// TwinCAT 3 PLC project PShEll_UniversalBlocks
// Title: PShEll Universal Blocks
// Company: Precision Systems Engineering
// Author: Control Systems Design Department
// ProjectVersion: 1.0.1.1
// Description: PSE Shell - Automation Software Development Kit
// ProgramVersion: 3.1.4023.0
// libraries:
//   CmpBitmapPool, * (System)
//   JS_MC_REF, * (Jenny Science AG)
//   Recipe Management, * (System)
//   Tc2_EtherCAT, * (Beckhoff Automation GmbH)
//   Tc2_IoFunctions, * (Beckhoff Automation GmbH)
//   Tc2_MC2, * (Beckhoff Automation GmbH)
//   Tc2_Standard, * (Beckhoff Automation GmbH)
//   Tc2_SUPS, * (Beckhoff Automation GmbH)
//   Tc2_System, * (Beckhoff Automation GmbH)
//   Tc2_SystemCX, * (Beckhoff Automation GmbH)
//   Tc2_TcpIp, * (Beckhoff Automation GmbH)
//   Tc2_Utilities, * (Beckhoff Automation GmbH)
//   Tc3_EventLogger, * (Beckhoff Automation GmbH)
//   Tc3_McCollisionAvoidance, * (Beckhoff Automation GmbH)
//   Tc3_McCompensations, * (Beckhoff Automation GmbH)
//   Tc3_McCoordinatedMotion, * (Beckhoff Automation GmbH)
//   Tc3_Module, * (Beckhoff Automation GmbH)
//   Tc3_XTS_Utility, * (Beckhoff Automation GmbH)
//   VisuDialogs, * (System)
//   VisuUserMgmt, * (System)
//   Tc2_Math,3.3.1.0,Beckhoff Automation GmbH
//   VisuSymbols,3.5.10.0,System
// project tree:
//   DUTs/Libs/Alarms/AlarmControler/ E_AlarmControlerState.TcDUT
//   DUTs/Libs/Alarms/VisuEvents/ E_EventType.TcDUT, ST_BaseEvent.TcDUT, ST_Event.TcDUT
//   DUTs/Libs/Axis/Universal Axis/ E_AxisJogDirection.TcDUT, E_AxisState.TcDUT, E_AxisStateInit.TcDUT, E_AxisStatePlcOpen.TcDUT
//   DUTs/Libs/Communication/TcpIp/ E_TcpIpDeviceState.TcDUT, E_TcpIpDeviceStateRecive.TcDUT, E_TcpIpDeviceStateSend.TcDUT, E_TcpIpServerStateRunning.TcDUT, ST_TcpBufferData.TcDUT
//   DUTs/Libs/Cylinder/Universal Cylinder/ E_CylinderError.TcDUT, E_CylinderState.TcDUT, E_CylinderStateGo.TcDUT
//   DUTs/Libs/Digital Devices/Digital Input/ E_DigitalInputExState.TcDUT
//   DUTs/Libs/Digital Devices/Lamp Indicator/ E_LampState.TcDUT
//   DUTs/Libs/Fixtures/UniversalFixture/ E_UniversalFixtureConnectionType.TcDUT, E_UniversalFixtureSampleResult.TcDUT, E_UniversalFixtureState.TcDUT, E_UniversalFixtureStateAbort.TcDUT, E_UniversalFixtureStateInit.TcDUT, E_UniversalFixtureStateMeasure.TcDUT, E_UniversalFixtureStateReset.TcDUT
//   DUTs/Libs/Platform/Common/ ST_UniversalPlatform.TcDUT
//   DUTs/Libs/Platform/Universal Machine/ E_MachineCtrlState.TcDUT
//   DUTs/Libs/Platform/Universal Safety/ E_SafetyCtrlState.TcDUT
//   DUTs/Libs/Platform/Universal Visu/ E_VisuCtrlAlarmControlState.TcDUT, E_VisuCtrlAxisImgType.TcDUT, E_VisuCtrlAxisJogMode.TcDUT, E_VisuCtrlCylinderImgType.TcDUT, E_VisuCtrlNavBarState.TcDUT, E_VisuCtrlPageState.TcDUT, E_VisuCtrlRecipeParameterType.TcDUT, E_VisuCtrlRecipesManagerState.TcDUT, E_VisuCtrlRobotImgType.TcDUT, E_VisuCtrlSingleAxisState.TcDUT, E_VisuCtrlSingleCylinderState.TcDUT, E_VisuCtrlSingleRobotState.TcDUT, E_VisuCtrUniversalMachineState.TcDUT, ST_VisuCtrlAxisFrame.TcDUT, ST_VisuCtrlCylinderFrame.TcDUT, ST_VisuCtrlFixtureFrame.TcDUT, ST_VisuCtrlInputFrame.TcDUT, ST_VisuCtrlOutputFrame.TcDUT, ST_VisuCtrlRecipeParameter.TcDUT, ST_VisuCtrlRecipesManager.TcDUT, ST_VisuCtrlRobotFrame.TcDUT, ST_VisuCtrlUnitFrame.TcDUT
//   DUTs/Libs/Robots/Mitsubishi/CR800/EtherCAT Registers/ ST_CR800EthercatData.TcDUT
//   DUTs/Libs/Robots/Mitsubishi/CR800/ E_CR800Error.TcDUT, ST_CR800UserDefinedArea.TcDUT
//   DUTs/Libs/Robots/Mitsubishi/CR800/StateMachine/ E_CR800State.TcDUT, E_CR800StateAborting.TcDUT, E_CR800StateCommandExchange.TcDUT, E_CR800StateCyclePausing.TcDUT, E_CR800StateCycleStopping.TcDUT, E_CR800StateDoingRequest.TcDUT, E_CR800StateHoming.TcDUT, E_CR800StateInitializing.TcDUT, E_CR800StateSendPosition.TcDUT
//   DUTs/Libs/Robots/Mitsubishi/ E_RobotActions.TcDUT, E_RobotSystemActions.TcDUT
//   DUTs/Libs/Utilities/CSV Data Exchanger/ E_CSVDataExchangerCountColumnsState.TcDUT, E_CSVDataExchangerInitState.TcDUT, E_CSVDataExchangerInsertIntoTableState.TcDUT, E_CSVDataExchangerSelectAllState.TcDUT, E_CSVDataExchangerSelectRowState.TcDUT, E_CSVDataExchangerSetNewPathState.TcDUT, E_CSVDataExchangerState.TcDUT, ST_CSV_Record.TcDUT
//   DUTs/Libs/Utilities/File Logger/ E_FileLoggerAddLogsState.TcDUT, E_FileLoggerInitState.TcDUT, E_FileLoggerSetNewPathState.TcDUT, E_FileLoggerState.TcDUT
//   DUTs/Libs/Utilities/Recipe Manager/ E_RecipesManagerReturns.TcDUT, E_RecipesManagerState.TcDUT, E_RecipesManagerStateBackup.TcDUT, E_RecipesManagerStateCreateRemove.TcDUT, E_RecipesManagerStateInit.TcDUT, E_RecipesManagerStateReload.TcDUT
//   DUTs/Libs/Utilities/TXT Data Exchanger/ E_TXTDataExchangerAddLogsState.TcDUT, E_TXTDataExchangerInitState.TcDUT, E_TXTDataExchangerSearchForFileState.TcDUT, E_TXTDataExchangerSetNewPathState.TcDUT, E_TXTDataExchangerState.TcDUT
//   DUTs/Libs/Vision/Cognex/ E_CognexCameraGetConnectionStatus.TcDUT, E_CognexCameraGetExprStatus.TcDUT, E_CognexCameraGetFileListStatus.TcDUT, E_CognexCameraGetFileStatus.TcDUT, E_CognexCameraGetJobStatus.TcDUT, E_CognexCameraGetOnlineStatus.TcDUT, E_CognexCameraGetPositionState.TcDUT, E_CognexCameraGetPositionStatus.TcDUT, E_CognexCameraGetValueEasyBuilderStatus.TcDUT, E_CognexCameraGetValueSpreadsheetStatus.TcDUT, E_CognexCameraGetValuesState.TcDUT, E_CognexCameraGetValuesStatus.TcDUT, E_CognexCameraGetValueStatus.TcDUT, E_CognexCameraImageTriggerStatus.TcDUT, E_CognexCameraInitState.TcDUT, E_CognexCameraLoadFileStatus.TcDUT, E_CognexCameraMethodState.TcDUT, E_CognexCameraPutLiveStatus.TcDUT, E_CognexCameraPutPortnumStatus.TcDUT, E_CognexCameraPutTimeoutStatus.TcDUT, E_CognexCameraPutUpdateStatus.TcDUT, E_CognexCameraPutWatchStatus.TcDUT, E_CognexCameraResetSystemStatus.TcDUT, E_CognexCameraSetJobStatus.TcDUT, E_CognexCameraSetOnlineStatus.TcDUT, E_CognexCameraState.TcDUT, E_CognexCameraStoreFileStatus.TcDUT
//   DUTs/Machine/Machine Control/ E_MachineCtrlStateInit.TcDUT, E_MachineCtrlStateUninitialized.TcDUT
//   DUTs/Machine/Shell API/ ST_Shell.TcDUT, ST_ShellFlags.TcDUT, ST_ShellPlatform.TcDUT, ST_ShellRecipeData.TcDUT
//   DUTs/Platform/Universal Visu/ ST_VisuCtrlRobotFrame.TcDUT (not stored)
//   / GlobalTextList.TcGTLO, Test.TcTTO, Visualization Manager.TcVMO (not stored), VISU_TASK.TcTTO
//   GVLs/ GVL.TcGVL
//   POUs/Libs/0_Checks/Checks/ CheckBounds.TcPOU, CheckDivDInt.TcPOU, CheckDivLInt.TcPOU, CheckDivLReal.TcPOU, CheckDivReal.TcPOU, CheckPointer.TcPOU, CheckRangeSigned.TcPOU, CheckRangeUnsigned.TcPOU, P_Checks.TcPOU
//   POUs/Libs/0_Checks/ GVL_Checks.TcGVL
//   POUs/Libs/Alarms/AlarmControler/ FB_AlarmControler.TcPOU, I_AlarmControler.TcIO
//   POUs/Libs/Alarms/VisuEvents/ FB_VisuEventsHandling.TcPOU, LDT_TO_STRING.TcPOU
//   POUs/Libs/Axis/ FB_AxisServo.TcPOU, FB_UniversalAxis.TcPOU, I_UniversalAxis.TcIO
//   POUs/Libs/Communication/TcpIp/ FUN_StringToTcpBufferData.TcPOU, FUN_TcpBufferDataToString.TcPOU
//   POUs/Libs/Communication/TcpIp/Tcp Buffer/ FB_TcpBuffer.TcPOU
//   POUs/Libs/Communication/TcpIp/Tcp Client/ FB_TcpClient.TcPOU
//   POUs/Libs/Communication/TcpIp/Tcp Device/ FB_TcpDevice.TcPOU, I_TcpDevice.TcIO
//   POUs/Libs/Communication/TcpIp/Tcp Server/ FB_TcpServer.TcPOU
//   POUs/Libs/Cylinder/Double Coil Cylinder/ FB_DoubleCoilCylinder.TcPOU, FB_DoubleCoilCylinder2.TcPOU
//   POUs/Libs/Cylinder/Single Coil Cylinder/ FB_SingleCoilCylinder.TcPOU, FB_SingleCoilCylinder2.TcPOU
//   POUs/Libs/Cylinder/Universal Cylinder/ FB_UniversalCylinder.TcPOU, I_UniversalCylinder.TcIO
//   POUs/Libs/Digital Devices/Digital Device/ FB_DigitalDevice.TcPOU, I_DigitalDevice.TcIO
//   POUs/Libs/Digital Devices/Digital Input/ FB_DigitalInput.TcPOU, FB_DigitalInputExt.TcPOU, I_DigitalInput.TcIO
//   POUs/Libs/Digital Devices/Digital Output/ FB_DigitalOutput.TcPOU, I_DigitalOutput.TcIO
//   POUs/Libs/Digital Devices/Lamp Indicator/ FB_Lamp.TcPOU, I_Lamp.TcIO
//   POUs/Libs/Fixtures/ FB_UniversalFixture.TcPOU, I_UniversalFixture.TcIO
//   POUs/Libs/Platform/Universal Machine/ FB_UniversalMachine.TcPOU, I_UniversalMachine.TcIO
//   POUs/Libs/Platform/Universal Safety/ FB_UniversalSafety.TcPOU, I_UniversalSafety.TcIO
//   POUs/Libs/Platform/Universal Visu/ FB_UniversalVisu.TcPOU, F_CloseDialog.TcPOU, F_OpenDialog.TcPOU
//   POUs/Libs/Robots/Mitsubishi/ FB_CR800EtherCAT.TcPOU, I_CR800EtherCAT.TcIO
//   POUs/Libs/Utilities/Beckhoff UPS/CX2xxx/ FB_UpsCx2xxx.TcPOU
//   POUs/Libs/Utilities/Beckhoff UPS/CX5xxx/ FB_UpsCx50xx.TcPOU, FB_UpsCx51xx.TcPOU, FB_UpsCx5xxx.TcPOU, I_BeckhoffUpsCX5xxx.TcIO
//   POUs/Libs/Utilities/Beckhoff UPS/Universal CX/ FB_UniversalCxUps.TcPOU, I_UniversalCxUps.TcIO
//   POUs/Libs/Utilities/CSV Data Exchanger/ FB_CSVDataExchanger.TcPOU, I_CSVDataExchanger.TcIO
//   POUs/Libs/Utilities/File Logger/ FB_FileLogger.TcPOU, I_FileLogger.TcIO
//   POUs/Libs/Utilities/Math/ FUN_Ceil.TcPOU
//   POUs/Libs/Utilities/Recipes Manager/ FB_RecipeParameter.TcPOU, FB_RecipesControler.TcPOU, I_RecipeParameter.TcIO, I_RecipesManager.TcIO
//   POUs/Libs/Utilities/StringMerge/ FUN_MergeLongStrings10.TcPOU, FUN_MergeStrings10.TcPOU, FUN_MergeStrings3.TcPOU, FUN_MergeStrings4.TcPOU, FUN_MergeStrings5.TcPOU, FUN_MergeStrings6.TcPOU
//   POUs/Libs/Utilities/Systemtime to String/ FUN_TimestructToDate.TcPOU, FUN_TimestructToTime.TcPOU
//   POUs/Libs/Utilities/TXT Data Exchanger/ FB_TXTDataExchanger.TcPOU, I_TXTDataExchanger.TcIO
//   POUs/Libs/Vision/Cognex/ FB_CognexCamera.TcPOU, I_CognexCamera.TcIO
//   POUs/Machine/Alarm Control/ PRG_AlarmControl.TcPOU
//   POUs/Machine/Machine Control/ FB_MachineControl.TcPOU, I_MachineControl.TcIO, PRG_MachineControl.TcPOU
//   POUs/Machine/Recipes Manager/ PRG_RecipesManager.TcPOU
//   POUs/Machine/Visu Control/ FB_VisuControl.TcPOU, F_CloseDialog_1.TcPOU, F_OpenDialog_1.TcPOU, PRG_VisuControl.TcPOU
//   VISUs/Alarms/ EventTable.TcVIS, EventTableNew.TcVIS (not stored), SingleEvent.TcVIS (not stored)
//   VISUs/Alarms/Image Pools/ IP_EventSeverity.TcIPO (not stored), IP_EventType.TcIPO (not stored)
//   VISUs/Alarms/Text Lists/ TL_EventServerity.TcTLO (not stored), TL_EventType.TcTLO (not stored)
//   VISUs/Headers/ Header.TcVIS, HeaderWinCE.TcVIS
//   VISUs/Headers/Image Pools/ IPHeader.TcIPO (not stored)
//   VISUs/Headers/Text Lists/ TL_HeaderMachineState.TcTLO
//   VISUs/ Main.TcVIS
//   VISUs/Manual/Image Pools/ IPAxis.TcIPO (not stored), IPCylinder.TcIPO (not stored), IPRobots.TcIPO (not stored)
//   VISUs/Manual/ SingleAxis.TcVIS, SingleFixture.TcVIS, SingleAxisJogInching.TcVIS, SingleAxisJogContinous.TcVIS, SingleAxisJogInchingModulo.TcVIS, SingleAxisJogStandardSlow.TcVIS, SingleAxisJogStandardFlast.TcVIS, SingleCylinder.TcVIS, SingleDigitalInput.TcVIS, SingleRobot.TcVIS, SingleSafeOutput.TcVIS (excluded from build), SingleSafeInput.TcVIS (excluded from build), SingleDigitalOutput.TcVIS
//   VISUs/Manual/Text Lists/ TL_ModeSwitchState.TcTLO, TL_SingleAxisJogMode.TcTLO, TL_SingleCylinderState.TcTLO, TL_SingleAxisState.TcTLO, TL_SingleRobotState.TcTLO
//   VISUs/Navigation/ NavBarAuto.TcVIS, NavBarAuxilary.TcVIS, NavBarEmpty.TcVIS, NavBarInitializing.TcVIS, NavBarManual.TcVIS, NavBarUninitialized.TcVIS, NavBarUtilities.TcVIS
//   VISUs/Pages/ PageInitializing.TcVIS, PageXtsEnviroment.TcVIS (excluded from build), PageAborting.TcVIS, PageAlarms.TcVIS, PageManualCylinders.TcVIS, PageManualRobots.TcVIS, PageManualInputs.TcVIS, PageManualAxis.TcVIS, PageManualOutputs.TcVIS, PageManualSafety.TcVIS (excluded from build), PageReadyInitialized.TcVIS, PageRecipesManager.TcVIS, PageReset.TcVIS, PageSwitchMode.TcVIS, PageXtsDiagnostic.TcVIS (excluded from build)
//   VISUs/Recipes/ SingleRecipesParameterTypeBool.TcVIS, SingleRecipesParameterTypeInteger.TcVIS, SingleRecipesParameterTypeReal.TcVIS, SingleRecipesParameterTypeString.TcVIS
//   VISUs/Recipes/Text Lists/ TL_RecipesManagerReturns.TcTLO, TL_RecipesManagerStatus.TcTLO
// real-time tasks:
//   TASK SampleTests Task: cycle T#10ms, priority 20, ADS port 350
//   TASK UniversalBlocks Task: cycle T#10ms, priority 22, ADS port 351
//   TASK Job Task: cycle default, priority 32
//   TASK VISU_TASK: cycle T#200000us, priority 30, ADS port 352
//   TASK XTS Task 1: cycle T#250us, priority 1, ADS port 353
//   TASK TestAlarms: cycle T#2ms, priority 21, ADS port 354
//   TASK Test: cycle T#10ms, priority 23, ADS port 355
// motion (NC):
//   TASK NC-Task 1 SAF: cycle T#2ms, priority 4, ADS port 501
//   TASK NC-Task 1 SVB: cycle T#10ms, priority 8, ADS port 511
//   AXIS Faulhaber_LM1247_PNP2_1 (id 11)
//     Dynamic: AccelerationMaximum=1000000, DecelerationMaximum=1000000, Acceleration=5000, Deceleration=5000, Jerk=10000
//     Velo: RefSearch=25, RefSync=15, SlowManual=10, FastManual=25
//     PositionAreaControl: Enable=false
//     TargetPosControl: Range=0.1, Time=0.01
//     OtherSettings: AllowMotionCmdToSlave=true, PulseDistancePos=10, PulseDistanceNeg=10
//     encoder EncType=19
//       EncPara: ScaleFactorNumerator=0.001, MaxCount=#xffffffff
//         SoftEndMinControl: Enable=true, Range=-80
//         SoftEndMaxControl: Enable=true, Range=80
//     drive DrvType=16
//       DrvPara: MaxCount=#xffffffff
//         Analog: VeloReferenz=2000, TorqueSetpointScale=10, ScaleFactorActTorque=0.1
//         TimeComp: TaskDelayCycles=1
//     controller CtrType=3
//       CtrPara: PriorControlFactor=1
//         PosDiffControl: Enable=false
//         PID: PosTn=0.1
//         Observer: BandWidth=20
//   AXIS Faulhaber_LM1247_PNP2_2 (id 7)
//     Dynamic: AccelerationMaximum=1000000, DecelerationMaximum=1000000, Acceleration=5000, Deceleration=5000, Jerk=10000
//     Velo: RefSearch=25, RefSync=15, SlowManual=10, FastManual=25
//     PositionAreaControl: Enable=false
//     TargetPosControl: Range=0.1, Time=0.01
//     OtherSettings: AllowMotionCmdToSlave=true, PulseDistancePos=10, PulseDistanceNeg=10
//     encoder EncType=19
//       EncPara: ScaleFactorNumerator=0.001, MaxCount=#xffffffff
//         SoftEndMinControl: Enable=true, Range=-80
//         SoftEndMaxControl: Enable=true, Range=80
//     drive DrvType=16
//       DrvPara: MaxCount=#xffffffff
//         Analog: VeloReferenz=2000, TorqueSetpointScale=10, ScaleFactorActTorque=0.1
//         TimeComp: TaskDelayCycles=1
//     controller CtrType=3
//       CtrPara: PriorControlFactor=1
//         PosDiffControl: Enable=false
//         PID: PosTn=0.1
//         Observer: BandWidth=20
//   AXIS Faulhaber_LM1247_PNP2_3 (id 8)
//     Dynamic: AccelerationMaximum=1000000, DecelerationMaximum=1000000, Acceleration=5000, Deceleration=5000, Jerk=10000
//     Velo: RefSearch=25, RefSync=15, SlowManual=10, FastManual=25
//     PositionAreaControl: Enable=false
//     TargetPosControl: Range=0.1, Time=0.01
//     OtherSettings: AllowMotionCmdToSlave=true, PulseDistancePos=10, PulseDistanceNeg=10
//     encoder EncType=19
//       EncPara: ScaleFactorNumerator=0.001, MaxCount=#xffffffff
//         SoftEndMinControl: Enable=true, Range=-80
//         SoftEndMaxControl: Enable=true, Range=80
//     drive DrvType=16
//       DrvPara: MaxCount=#xffffffff
//         Analog: VeloReferenz=2000, TorqueSetpointScale=10, ScaleFactorActTorque=0.1
//         TimeComp: TaskDelayCycles=1
//     controller CtrType=3
//       CtrPara: PriorControlFactor=1
//         PosDiffControl: Enable=false
//         PID: PosTn=0.1
//         Observer: BandWidth=20
//   AXIS Faulhaber_LM1247_PNP2_4 (id 9)
//     Dynamic: AccelerationMaximum=1000000, DecelerationMaximum=1000000, Acceleration=5000, Deceleration=5000, Jerk=10000
//     Velo: RefSearch=25, RefSync=15, SlowManual=10, FastManual=25
//     PositionAreaControl: Enable=false
//     TargetPosControl: Range=0.1, Time=0.01
//     OtherSettings: AllowMotionCmdToSlave=true, PulseDistancePos=10, PulseDistanceNeg=10
//     encoder EncType=19
//       EncPara: ScaleFactorNumerator=0.001, MaxCount=#xffffffff
//         SoftEndMinControl: Enable=true, Range=-80
//         SoftEndMaxControl: Enable=true, Range=80
//     drive DrvType=16
//       DrvPara: MaxCount=#xffffffff
//         Analog: VeloReferenz=2000, TorqueSetpointScale=10, ScaleFactorActTorque=0.1
//         TimeComp: TaskDelayCycles=1
//     controller CtrType=3
//       CtrPara: PriorControlFactor=1
//         PosDiffControl: Enable=false
//         PID: PosTn=0.1
//         Observer: BandWidth=20
//   AXIS Faulhaber_LM1247_PNP2_5 (id 10)
//     Dynamic: AccelerationMaximum=1000000, DecelerationMaximum=1000000, Acceleration=5000, Deceleration=5000, Jerk=10000
//     Velo: RefSearch=25, RefSync=15, SlowManual=10, FastManual=25
//     PositionAreaControl: Enable=false
//     TargetPosControl: Range=0.1, Time=0.01
//     OtherSettings: AllowMotionCmdToSlave=true, PulseDistancePos=10, PulseDistanceNeg=10
//     encoder EncType=19
//       EncPara: ScaleFactorNumerator=0.001, MaxCount=#xffffffff
//         SoftEndMinControl: Enable=true, Range=-80
//         SoftEndMaxControl: Enable=true, Range=80
//     drive DrvType=16
//       DrvPara: MaxCount=#xffffffff
//         Analog: VeloReferenz=2000, TorqueSetpointScale=10, ScaleFactorActTorque=0.1
//         TimeComp: TaskDelayCycles=1
//     controller CtrType=3
//       CtrPara: PriorControlFactor=1
//         PosDiffControl: Enable=false
//         PID: PosTn=0.1
//         Observer: BandWidth=20
//   AXIS Faulhaber_LM1247_PNP2_6 (id 12)
//     Dynamic: AccelerationMaximum=1000000, DecelerationMaximum=1000000, Acceleration=5000, Deceleration=5000, Jerk=10000
//     Velo: RefSearch=25, RefSync=15, SlowManual=10, FastManual=25
//     PositionAreaControl: Enable=false
//     TargetPosControl: Range=0.1, Time=0.01
//     OtherSettings: AllowMotionCmdToSlave=true, PulseDistancePos=10, PulseDistanceNeg=10
//     encoder EncType=19
//       EncPara: ScaleFactorNumerator=0.001, MaxCount=#xffffffff
//         SoftEndMinControl: Enable=true, Range=-80
//         SoftEndMaxControl: Enable=true, Range=80
//     drive DrvType=16
//       DrvPara: MaxCount=#xffffffff
//         Analog: VeloReferenz=2000, TorqueSetpointScale=10, ScaleFactorActTorque=0.1
//         TimeComp: TaskDelayCycles=1
//     controller CtrType=3
//       CtrPara: PriorControlFactor=1
//         PosDiffControl: Enable=false
//         PID: PosTn=0.1
//         Observer: BandWidth=20
//   AXIS Faulhaber_LM1247_PNP1_2 (id 14)
//     Dynamic: AccelerationMaximum=1000000, DecelerationMaximum=1000000, Acceleration=5000, Deceleration=5000, Jerk=10000
//     Velo: RefSearch=25, RefSync=25, SlowManual=10, FastManual=25
//     PositionAreaControl: Enable=false
//     TargetPosControl: Range=0.1, Time=0.01
//     OtherSettings: AllowMotionCmdToSlave=true, PulseDistancePos=10, PulseDistanceNeg=10
//     encoder EncType=19
//       EncPara: ScaleFactorNumerator=0.001, MaxCount=#xffffffff
//         SoftEndMinControl: Enable=true, Range=-80
//         SoftEndMaxControl: Enable=true, Range=80
//     drive DrvType=16
//       DrvPara: MaxCount=#xffffffff
//         Analog: VeloReferenz=2000, TorqueSetpointScale=10, ScaleFactorActTorque=0.1
//         TimeComp: TaskDelayCycles=1
//     controller CtrType=3
//       CtrPara: PriorControlFactor=1
//         PosDiffControl: Enable=false
//         PID: PosTn=0.1
//         Observer: BandWidth=20
//   AXIS Faulhaber_LM1247_PNP1_6 (id 13)
//     Dynamic: AccelerationMaximum=1000000, DecelerationMaximum=1000000, Acceleration=5000, Deceleration=5000, Jerk=10000
//     Velo: RefSearch=25, RefSync=25, SlowManual=10, FastManual=25
//     PositionAreaControl: Enable=false
//     TargetPosControl: Range=0.1, Time=0.01
//     OtherSettings: AllowMotionCmdToSlave=true, PulseDistancePos=10, PulseDistanceNeg=10
//     encoder EncType=1
//       EncPara: ScaleFactorNumerator=0.001
//         SoftEndMinControl: Enable=true, Range=-80
//         SoftEndMaxControl: Enable=true, Range=80
//     drive DrvType=5
//       Analog: VeloReferenz=10, TorqueSetpointScale=10, ScaleFactorActTorque=0.1
//       TimeComp: TaskDelayCycles=1
//     controller CtrType=3
//       CtrPara: PriorControlFactor=1
//         PosDiffControl: Enable=false
//         PID: PosTn=0.1
//         Observer: BandWidth=20
//   AXIS Mover Axis 1 (id 15)
//     General: UnitFlags=#x00000004
//     Dynamic: AccelerationMaximum=80000, DecelerationMaximum=80000, Acceleration=20000, Deceleration=20000, Jerk=200000
//     Velo: Maximum=4000
//     PositionAreaControl: Enable=false
//     TargetPosControl: Enable=false
//     OtherSettings: AllowMotionCmdToSlave=true, AllowMotionCmdToExtSetGenAxis=true
//     encoder EncType=28
//       EncPara: ModuloFactor=2500, ToleranceWndModuloStart=0.2, MaxCount=#xffffffff
//     drive DrvType=22
//       DrvPara: MaxCount=#xffffffff, DriveControlDWord=#x00000100
//         Analog: VeloReferenz=4200, TorqueSetpointScale=10
//         TimeComp: TaskDelayCycles=1
//     controller CtrType=1
//       CtrPara: PriorControlFactor=1
//         PosDiffControl: Range=10
//         Observer: BandWidth=20
//   AXIS Mover Axis 2 (id 16)
//     General: UnitFlags=#x00000004
//     Dynamic: AccelerationMaximum=80000, DecelerationMaximum=80000, Acceleration=20000, Deceleration=20000, Jerk=200000
//     Velo: Maximum=4000
//     PositionAreaControl: Enable=false
//     TargetPosControl: Enable=false
//     OtherSettings: AllowMotionCmdToSlave=true, AllowMotionCmdToExtSetGenAxis=true
//     encoder EncType=28
//       EncPara: ModuloFactor=2500, ToleranceWndModuloStart=0.2, MaxCount=#xffffffff
//     drive DrvType=22
//       DrvPara: MaxCount=#xffffffff, DriveControlDWord=#x00000100
//         Analog: VeloReferenz=4200, TorqueSetpointScale=10
//         TimeComp: TaskDelayCycles=1
//     controller CtrType=1
//       CtrPara: PriorControlFactor=1
//         PosDiffControl: Range=10
//         Observer: BandWidth=20
//   AXIS Mover Axis 3 (id 17)
//     General: UnitFlags=#x00000004
//     Dynamic: AccelerationMaximum=80000, DecelerationMaximum=80000, Acceleration=20000, Deceleration=20000, Jerk=200000
//     Velo: Maximum=4000
//     PositionAreaControl: Enable=false
//     TargetPosControl: Enable=false
//     OtherSettings: AllowMotionCmdToSlave=true, AllowMotionCmdToExtSetGenAxis=true
//     encoder EncType=28
//       EncPara: ModuloFactor=2500, ToleranceWndModuloStart=0.2, MaxCount=#xffffffff
//     drive DrvType=22
//       DrvPara: MaxCount=#xffffffff, DriveControlDWord=#x00000100
//         Analog: VeloReferenz=4200, TorqueSetpointScale=10
//         TimeComp: TaskDelayCycles=1
//     controller CtrType=1
//       CtrPara: PriorControlFactor=1
//         PosDiffControl: Range=10
//         Observer: BandWidth=20
//   AXIS Mover Axis 4 (id 18)
//     General: UnitFlags=#x00000004
//     Dynamic: AccelerationMaximum=80000, DecelerationMaximum=80000, Acceleration=20000, Deceleration=20000, Jerk=200000
//     Velo: Maximum=4000
//     PositionAreaControl: Enable=false
//     TargetPosControl: Enable=false
//     OtherSettings: AllowMotionCmdToSlave=true, AllowMotionCmdToExtSetGenAxis=true
//     encoder EncType=28
//       EncPara: ModuloFactor=2500, ToleranceWndModuloStart=0.2, MaxCount=#xffffffff
//     drive DrvType=22
//       DrvPara: MaxCount=#xffffffff, DriveControlDWord=#x00000100
//         Analog: VeloReferenz=4200, TorqueSetpointScale=10
//         TimeComp: TaskDelayCycles=1
//     controller CtrType=1
//       CtrPara: PriorControlFactor=1
//         PosDiffControl: Range=10
//         Observer: BandWidth=20
//   AXIS Mover Axis 5 (id 19)
//     General: UnitFlags=#x00000004
//     Dynamic: AccelerationMaximum=80000, DecelerationMaximum=80000, Acceleration=20000, Deceleration=20000, Jerk=200000
//     Velo: Maximum=4000
//     PositionAreaControl: Enable=false
//     TargetPosControl: Enable=false
//     OtherSettings: AllowMotionCmdToSlave=true, AllowMotionCmdToExtSetGenAxis=true
//     encoder EncType=28
//       EncPara: ModuloFactor=2500, ToleranceWndModuloStart=0.2, MaxCount=#xffffffff
//     drive DrvType=22
//       DrvPara: MaxCount=#xffffffff, DriveControlDWord=#x00000100
//         Analog: VeloReferenz=4200, TorqueSetpointScale=10
//         TimeComp: TaskDelayCycles=1
//     controller CtrType=1
//       CtrPara: PriorControlFactor=1
//         PosDiffControl: Range=10
//         Observer: BandWidth=20
//   AXIS Mover Axis 6 (id 20)
//     General: UnitFlags=#x00000004
//     Dynamic: AccelerationMaximum=80000, DecelerationMaximum=80000, Acceleration=20000, Deceleration=20000, Jerk=200000
//     Velo: Maximum=4000
//     PositionAreaControl: Enable=false
//     TargetPosControl: Enable=false
//     OtherSettings: AllowMotionCmdToSlave=true, AllowMotionCmdToExtSetGenAxis=true
//     encoder EncType=28
//       EncPara: ModuloFactor=2500, ToleranceWndModuloStart=0.2, MaxCount=#xffffffff
//     drive DrvType=22
//       DrvPara: MaxCount=#xffffffff, DriveControlDWord=#x00000100
//         Analog: VeloReferenz=4200, TorqueSetpointScale=10
//         TimeComp: TaskDelayCycles=1
//     controller CtrType=1
//       CtrPara: PriorControlFactor=1
//         PosDiffControl: Range=10
//         Observer: BandWidth=20
//   AXIS OnlineSimulationAxis (id 6)
//     General: UnitName=m
//     Dynamic: Acceleration=4.31553, Deceleration=4.31553, Jerk=0.1
//     Velo: SlowManual=125, FastManual=425, Maximum=45540
//     OtherSettings: AllowMotionCmdToSlave=true
//     encoder EncType=1
//     drive DrvType=5
//       Analog: VeloReferenz=1000000000000, TorqueSetpointScale=10, ScaleFactorActTorque=0.1
//       TimeComp: TaskDelayCycles=1
//     controller CtrType=1
//       CtrPara: PriorControlFactor=1
//         Observer: BandWidth=20
//   AXIS OnlineSimulationAxisCA1 (id 1)
//     General: UnitName=Degree
//     OtherSettings: AllowMotionCmdToSlave=true, AllowMotionCmdToExtSetGenAxis=true
//     encoder EncType=1
//     drive DrvType=5
//       Analog: TorqueSetpointScale=10, ScaleFactorActTorque=0.1
//       TimeComp: TaskDelayCycles=1
//     controller CtrType=1
//       CtrPara: PriorControlFactor=1
//         Observer: BandWidth=20
//   AXIS OnlineSimulationAxisCA2 (id 3)
//     General: UnitName=Degree
//     OtherSettings: AllowMotionCmdToSlave=true, AllowMotionCmdToExtSetGenAxis=true
//     encoder EncType=1
//     drive DrvType=5
//       Analog: TorqueSetpointScale=10, ScaleFactorActTorque=0.1
//       TimeComp: TaskDelayCycles=1
//     controller CtrType=1
//       CtrPara: PriorControlFactor=1
//         Observer: BandWidth=20
//   AXIS BeckhoffServoAxis (id 2)
//     General: UnitName=Degree
//     Dynamic: Acceleration=21843, Deceleration=21843, Jerk=65529
//     Velo: RefSearch=145.62, RefSync=145.62, SlowManual=728.1, FastManual=4368.6, Fast=14562, Maximum=14562
//     OtherSettings: AllowMotionCmdToSlave=true
//     encoder EncType=19
//       EncPara: ScaleFactorNumerator=360, ScaleFactorDenominator=1048576, MaxCount=#xffffffff
//     drive DrvType=16
//       DrvPara: MaxCount=#xffffffff
//         Analog: VeloReferenz=16018.2, VeloScale=32, TorqueSetpointScale=10, ScaleFactorActTorque=0.1
//         TimeComp: TaskDelayCycles=1
//     controller CtrType=1
//       CtrPara: PriorControlFactor=1
//         PID: PosKp=10
//         Observer: BandWidth=20
//   AXIS JennyScienceAxisX (id 4)
//     Velo: SlowManual=5, FastManual=30, Maximum=4500
//     OtherSettings: AllowMotionCmdToSlave=true
//     encoder EncType=19
//       EncPara: ScaleFactorNumerator=0.001, MaxCount=#xffffffff
//         SoftEndMinControl: Enable=true
//         SoftEndMaxControl: Enable=true, Range=320
//     drive DrvType=16
//       DrvPara: MaxCount=#xffffffff, DriveControlDWord=#x00000100
//         Analog: VeloReferenz=4500, TorqueSetpointScale=10, ScaleFactorActTorque=0.1
//         TimeComp: TaskDelayCycles=1
//     controller CtrType=9
//       CtrPara: PriorControlFactor=1
//         PosDiffControl: Enable=false
//         Observer: BandWidth=20
//   AXIS JennyScienceAxisZ (id 5)
//     Velo: SlowManual=5, FastManual=30, Maximum=4500
//     OtherSettings: AllowMotionCmdToSlave=true
//     encoder EncType=19
//       EncPara: ScaleFactorNumerator=0.001, MaxCount=#xffffffff
//     drive DrvType=16
//       DrvPara: MaxCount=#xffffffff, DriveControlDWord=#x00000100
//         Analog: VeloReferenz=4500, TorqueSetpointScale=10, ScaleFactorActTorque=0.1
//         TimeComp: TaskDelayCycles=1
//     controller CtrType=9
//       CtrPara: PriorControlFactor=1
//         PosDiffControl: Enable=false
//         Observer: BandWidth=20
// variable links:
//   NC-Task 1 SAF/Axes/Mover Axis 1 <-> TcCOM Objects/XtsProcessingUnit 1/Mover 1
//     SoftDrive 15/Data Pointer/InputPointer1 <-> Inputs/SoftDriveInput
//     SoftDrive 15/Data Pointer/OutputPointer1 <-> Outputs/SoftDriveOutput
//   NC-Task 1 SAF/Axes/Mover Axis 2 <-> TcCOM Objects/XtsProcessingUnit 1/Mover 2
//     SoftDrive 16/Data Pointer/InputPointer1 <-> Inputs/SoftDriveInput
//     SoftDrive 16/Data Pointer/OutputPointer1 <-> Outputs/SoftDriveOutput

CONFIGURATION PShEll_UniversalBlocks
    RESOURCE PLC ON TwinCAT3
        TASK Test(INTERVAL := T#10ms, PRIORITY := 23);
        TASK VISU_TASK(INTERVAL := T#100us, PRIORITY := 30);
        PROGRAM PRG_AlarmControl WITH Test : PRG_AlarmControl;
        PROGRAM PRG_MachineControl WITH Test : PRG_MachineControl;
        PROGRAM PRG_RecipesManager WITH Test : PRG_RecipesManager;
        PROGRAM PRG_VisuControl WITH Test : PRG_VisuControl;
        PROGRAM VisuElems_Visu_Prg WITH VISU_TASK : VisuElems.Visu_Prg;
    END_RESOURCE
END_CONFIGURATION

// ---- DUTs/Libs/Alarms/AlarmControler/E_AlarmControlerState.TcDUT
{attribute 'strict'}
TYPE E_AlarmControlerState :
(
	ALARM_CONTROLER_UNINITIALIZED 		:= 0,
	ALARM_CONTROLER_INITIALIZING		:= 10,
	ALARM_CONTROLER_READY_INITIALIZED	:= 20,
	ALARM_CONTROLER_IDLE				:= 30,
	ALARM_CONTROLER_CONFIRM_ALL			:= 40,
	ALARM_CONTROLER_CONFIRM_ALL_DONE	:= 50,
	ALARM_CONTROLER_CLEAR_ALL			:= 60,
	ALARM_CONTROLER_CLEAR_ALL_DONE		:= 70,
	ALARM_CONTROLER_CONFIRM				:= 80,
	ALARM_CONTROLER_CONFIRM_DONE		:= 90,
	ALARM_CONTROLER_CLEAR				:= 100,
	ALARM_CONTROLER_CLEAR_DONE			:= 110,
	ALARM_CONTROLER_EXPORT				:= 120,
	ALARM_CONTROLER_EXPORT_DONE			:= 130,
	ALARM_CONTROLER_ABORTING 			:= -10
);
END_TYPE

// ---- DUTs/Libs/Alarms/VisuEvents/E_EventType.TcDUT
{attribute 'qualified_only'}
{attribute 'strict'}
TYPE E_EventType :
(
	EMPTY			:= 0,
	ALARM_RAISED 	:= 10,
	ALARM_CONFIRMED	:= 20,
	ALARM_CLEARED	:= 30,
	MESSAGE			:= 40
);
END_TYPE

// ---- DUTs/Libs/Alarms/VisuEvents/ST_BaseEvent.TcDUT
TYPE ST_BaseEvent :
STRUCT
	guidEventClass 			: 	GUID;														(*  *)
	eSeverity 				: 	TcEventSeverity;											(*  *)
	iEventId				:	UDINT;														(* Event ID number *)
	iTimeStamp				: 	ULINT;														(* Timestamp when the event occured *)
	sJsonAttribute	 		: 	STRING (10000);												(* Additional parameters *)
	sSourceName				:	STRING(Tc3_EventLogger.ParameterList.cSourceNameSize-1);	(**)
	iTcArguments			: 	I_TcArguments;												(**)
	eEventType				:	E_EventType;												(**)
	iType					:	BYTE;														(* 1 -> Alarm, 2 -> Message*)
	iSourceID				:	UDINT;														(**)
END_STRUCT
END_TYPE

// ---- DUTs/Libs/Alarms/VisuEvents/ST_Event.TcDUT
TYPE ST_Event :
STRUCT
	iType					:	BYTE;					//1 -> Alarm, 2 -> message
	eSeverity 				: 	TcEventSeverity;		//typ zdarzenia
	iEventId				:	UDINT;					//ID zdarzenia
	iTimeStamp				: 	ULINT;					//stempel zdarzenia
	iTimeStampConfirmed		: 	ULINT;					//stempel zdarzenia
	iTimeStampCleared		: 	ULINT;					//stempel zdarzenia	
	sJsonAttribute 			: 	STRING (10000);			//parametry dodatkowe						//teks eventu z tlumaczniem
	sEventText				:	STRING(255);
	guidEventClass 			: 	GUID;
	sSourceName				:	STRING(Tc3_EventLogger.ParameterList.cSourceNameSize-1);
	iSourceID				:	UDINT;
END_STRUCT
END_TYPE

// ---- DUTs/Libs/Axis/Universal Axis/E_AxisJogDirection.TcDUT
{attribute 'strict'}
TYPE E_AxisJogDirection :
(
	AXIS_JOG_DIR_POSITIVE := 0,	(* Perform jog in positive direction *)
	AXIS_JOG_DIR_NEGATIVE := 10	(* Perform jog in negative direction *)
);
END_TYPE

// ---- DUTs/Libs/Axis/Universal Axis/E_AxisState.TcDUT
{attribute 'strict'}
TYPE E_AxisState :
(
	AXIS_UNINITIALIZED		:= 0,	(* Axis is not prepared to work - power is off *)
	AXIS_INITIALIZING		:= 10,	(* Axis is preparing to power - reset FB and power on *)
	AXIS_READY_INITIALIZED	:= 20,	(*  *)
	AXIS_IDLE				:= 30,	(* Axis is ready for orders *)
	AXIS_HOME				:= 40,	(* Axis is homing to reference point *)
	AXIS_HOME_DONE			:= 50,	(* Axis homing procedure has finished - fererence position has been found *)
	AXIS_MOVE_VELOCITY		:= 60,	(* Axis started continous motion to setpoint velocity - accelerating *)
	AXIS_MOVE_VELOCITY_DONE	:= 70,	(* Axis reached constant setpoint velocity for continous motion *)
	AXIS_MOVE_ABSOLUTE		:= 80,	(* Axis is moving to absolute position - discrete motion *)
	AXIS_MOVE_ABSOLUTE_DONE	:= 90,	(* Axis movement to absolute position finished *)
	AXIS_MOVE_ADDITIVE		:= 100,	(* Axis relative movement by desired distance *)
	AXIS_MOVE_ADDITIVE_DONE	:= 110,	(* Axis relative relative movement by desired distance finished *)
	AXIS_MOVE_RELATIVE		:= 120,	(* Axis relative movement by desired distance *)
	AXIS_MOVE_RELATIVE_DONE	:= 130,	(* Axis relative relative movement by desired distance finished *)
	AXIS_MOVE_JOG			:= 140,	(* Axis manual move using jog function *)
	AXIS_MOVE_JOG_DONE		:= 150,	(* Axis jog done *)
	AXIS_STOP				:= 160,	(* Axis is stopping *)
	AXIS_STOP_DONE			:= 170,	(* Axis stopped *)
	AXIS_HALT				:= 180,	(* Axis halts started motion command *)
	AXIS_HALT_DONE			:= 190,	(* Axis motion halted *)
	AXIS_RESET				:= 200,	(* Axis is resseting all function blocks and occured errors *)
	AXIS_RESET_DONE			:= 210,	(* Axis reset procedure done *)
	AXIS_COUPLE				:= 220, (* Axis is synchronizing to another master axis *)
	AXIS_COUPLE_DONE		:= 230,	(* Axis coupled to another master axis*)
	AXIS_DECOUPLE			:= 240,	(* Axis is decoupling from synchronized motion *)
	AXIS_DECOUPLE_DONE		:= 250,	(* Axis decoupled from synchronizing motion*)
	AXIS_UNLOCK				:= 260,	(* Axis is unlocking after stop command *)
	AXIS_UNLOCK_DONE		:= 270,	(* Axis unlocked after stop command *)
	AXIS_EXTENSION			:= 999,	(* Special state used by child FB's to implement additional states *)
	AXIS_ABORTING			:= -10	(* Aborting *)
);
END_TYPE

// ---- DUTs/Libs/Axis/Universal Axis/E_AxisStateInit.TcDUT
{attribute 'strict'}
TYPE E_AxisStateInit :
(
	AXIS_INIT_RESET		:= 0,	(* Reseting all function blocks *)
	AXIS_INIT_POWER_ON	:= 10,	(* Powering on the axis *)
	AXIS_INIT_DONE		:= 20	(* Initialization done *)
);
END_TYPE

// ---- DUTs/Libs/Axis/Universal Axis/E_AxisStatePlcOpen.TcDUT
{attribute 'strict'}
TYPE E_AxisStatePlcOpen :
(
	AXIS_PLCOPEN_DISABLED				:= 0,	(* Axis power controler if of *)
	AXIS_PLCOPEN_STANDSTILL				:= 10,	(* Axis is powered on *)
	AXIS_PLCOPEN_HOMING					:= 20,	(* Axis performs homing procedure *)
	AXIS_PLCOPEN_STOPPING				:= 30,	(* Axis is stopping the movement *)
	AXIS_PLCOPEN_CONTINUOUS_MOTION		:= 40,	(* Axis is moving continuosly with constant speed *)
	AXIS_PLCOPEN_DISCRETE_MOTION		:= 50,	(* Axis is moving from point to point *)
	AXIS_PLCOPEN_SYNCHRONIZED_MOTION 	:= 60,	(* Axis is moving in synchronized motion to master *)
	AXIS_PLCOPEN_ERRORSTOP				:= 70	(* Axis stoped because of error *)
);
END_TYPE

// ---- DUTs/Libs/Communication/TcpIp/E_TcpIpDeviceState.TcDUT
{attribute 'strict'}
TYPE E_TcpIpDeviceState :
(
	TCPIP_DEVICE_UNINITIALIZED 		:= 0,	(* Function block not ready to work - disconnected *)
	TCPIP_DEVICE_INITIALIZING		:= 10,	(* TCP/IP client creating client socket / TCP/IP server creating listener socket *)
	TCPIP_DEVICE_READY_INITIALIZED	:= 20,	(* Initialization finieshed successfull *)
	TCPIP_DEVICE_RUNNING			:= 30,	(* TCP/IP client data exchange with server / TCP/IP server listening for clients or data exchange with client *)
	TCPIP_DEVICE_ABORTING			:= -10	(* Closing connection and deinitialization of function block *)
);
END_TYPE

// ---- DUTs/Libs/Communication/TcpIp/E_TcpIpDeviceStateRecive.TcDUT
{attribute 'strict'}
TYPE E_TcpIpDeviceStateRecive :
(
	TCPIP_DEVICE_DATA_EXCHANGE_GET_RECIVED_DATA := 0,	(* Starting data reciving *)
	TCPIP_DEVICE_DATA_EXCHANGE_RECIVE_DONE		:= 10,	(* Waiting for any data form server *)
	TCPIP_DEVICE_DATA_EXCHANGE_WRITE_TO_BUFFER  := 20	
);
END_TYPE

// ---- DUTs/Libs/Communication/TcpIp/E_TcpIpDeviceStateSend.TcDUT
{attribute 'strict'}
TYPE E_TcpIpDeviceStateSend :
(
	TCPIP_DEVICE_DATA_EXCHANGE_GET_SEND_DATA	:= 0,	(* Append send data to clear send buffer *)
	TCPIP_DEVICE_DATA_EXCHANGE_SEND				:= 10,	(* Send data to server*)
	TCPIP_DEVICE_DATA_EXCHANGE_SEND_DONE		:= 20
);
END_TYPE

// ---- DUTs/Libs/Communication/TcpIp/E_TcpIpServerStateRunning.TcDUT
{attribute 'strict'}
TYPE E_TcpIpServerStateRunning :
(
	TCPIP_SERVER_RUNNING_START_LISTENING 		:= 0,	(* Re/Starting connection procedure *)
	TCPIP_SERVER_RUNNING_WAIT_FOR_CONNECTION	:= 10,	(* Waiting for any client *)
	TCPIP_SERVER_RUNNING_DATA_EXCHANGE 			:= 20,	(* Exchanging data with connected client *)
	TCPIP_SERVER_RUNNING_CLOSE_CONNECTION 		:= 30,	(* Closing current connection on request *)
	TCPIP_SERVER_RUNNING_CLOSE_CONNECTION_DONE	:= 40	(* Connection closed *)
);
END_TYPE

// ---- DUTs/Libs/Communication/TcpIp/ST_TcpBufferData.TcDUT
TYPE ST_TcpBufferData :
STRUCT
	arrData : ARRAY[1..8192] OF BYTE;
	iLength : UDINT;
END_STRUCT
END_TYPE

// ---- DUTs/Libs/Cylinder/Universal Cylinder/E_CylinderError.TcDUT
{attribute 'strict'}
TYPE E_CylinderError :
(
	CYLINDER_ERROR_OK						:= 0,	(*  *)
	CYLINDER_ERROR_MOVE_HOME_TIMED_OUT 		:= 10,	(*  *)
	CYLINDER_ERROR_MOVE_ACTIVE_TIMED_OUT 	:= 20	(*  *)
);
END_TYPE

// ---- DUTs/Libs/Cylinder/Universal Cylinder/E_CylinderState.TcDUT
{attribute 'strict'}
TYPE E_CylinderState :
(
	CYLINDER_UNINITIALIZED		:= 0,	(* Cylinder is uninitialized *)
	CYLINDER_INITIALIZING		:= 10,	(* Initialization in progress *)
	CYLINDER_READY_INITIALIZED	:= 20,	(*  *)
	CYLINDER_IDLE				:= 30,	(* Cylinder ready to work *)
	CYLINDER_GO_ACTIVE			:= 40,	(* Cylinder is going to active position *)
	CYLINDER_GO_ACTIVE_DONE		:= 50,	(* Cylinder is in active position *)
	CYLINDER_GO_HOME			:= 60,	(* Cylinder is going to home position *)
	CYLINDER_GO_HOME_DONE		:= 70,	(* Cylinder is in home position *)
	CYLINDER_RELEASE			:= 80,	(* Cylinder is going to release all valves *)
	CYLINDER_RELEASE_DONE		:= 90,	(* Cylinder has been released *)
	CYLINDER_RESET				:= 100,	(* Reseting function block *)
	CYLINDER_RESET_DONE			:= 110,	(* Reset done *)
	CYLINDER_ABORTING 			:= -10	(* Aborting *)
);
END_TYPE

// ---- DUTs/Libs/Cylinder/Universal Cylinder/E_CylinderStateGo.TcDUT
{attribute 'strict'}
TYPE E_CylinderStateGo :
(
	CYLINDER_MOVE_START_TRACKING	:= 0,
	CYLINDER_MOVE_DELAY				:= 10,
	CYLINDER_MOVE_DONE				:= 20
);
END_TYPE

// ---- DUTs/Libs/Digital Devices/Digital Input/E_DigitalInputExState.TcDUT
{attribute 'strict'}
TYPE E_DigitalInputExState :
(
	DIGITAL_INPUT_EX_UNINITIALIZED			:= 0,	(*  *)
	DIGITAL_INPUT_EX_INITIALIZING			:= 10,	(*  *)
	DIGITAL_INPUT_EX_READY_INITIALIZED		:= 20,	(*  *)
	DIGITAL_INPUT_EX_IDLE					:= 30,	(*  *)
	DIGITAL_INPUT_EX_TIMEOUT_TRACKING		:= 40,	(*  *)
	DIGITAL_INPUT_EX_TIMEOUT_TRACKING_DONE	:= 50,	(*  *)
	DIGITAL_INPUT_EX_RESET					:= 60,	(*  *)
	DIGITAL_INPUT_EX_RESET_DONE				:= 70,	(*  *)
	DIGITAL_INPUT_EX_ABORTING				:= -10	(*  *)
);
END_TYPE

// ---- DUTs/Libs/Digital Devices/Lamp Indicator/E_LampState.TcDUT
{attribute 'strict'}
TYPE E_LampState :
(
	LAMP_OFF 			:= 0,	(* Lamp is off *)
	LAMP_ON				:= 10,	(* Lamp is on *)
	LAMP_BLINKING_OFF	:= 20,	(* Lamp is blinking - current off *)
	LAMP_BLINKING_ON	:= 30	(* Lamp is bliniking - current on *)
);
END_TYPE

// ---- DUTs/Libs/Fixtures/UniversalFixture/E_UniversalFixtureConnectionType.TcDUT
{attribute 'strict'}
TYPE E_UniversalFixtureConnectionType :
(
	UNIVERSAL_FIXTURE_CLIENT_CONNECTION		:= 0,	(* Fixture will connect as a client *)
	UNIVERSAL_FIXTURE_SERVER_CONNECTION 	:= 10	(* Fixture will connect as a server  *)
);
END_TYPE

// ---- DUTs/Libs/Fixtures/UniversalFixture/E_UniversalFixtureSampleResult.TcDUT
{attribute 'strict'}
TYPE E_UniversalFixtureSampleResult :
(
	UNIVERSAL_FIXTURE_SAMPLE_REJECTED 	:= 0,	(* Sample didn't meet the requierments *)
	UNIVERSAL_FIXTURE_SAMPLE_ACCEPTED 	:= 10,	(*  *)
	UNIVERSAL_FIXTURE_SAMPLE_UNKNOWN	:= 20	(*  *)
);
END_TYPE

// ---- DUTs/Libs/Fixtures/UniversalFixture/E_UniversalFixtureState.TcDUT
{attribute 'strict'}
TYPE E_UniversalFixtureState :
(
	UNIVERSAL_FIXTURE_UNINITIALIZED 	:= 0,	(*  *)
	UNIVERSAL_FIXTURE_INITIALIZING 		:= 10,	(*  *)
	UNIVERSAL_FIXTURE_READY 			:= 20,	(*  *)
	UNIVERSAL_FIXTURE_IDLE				:= 30,	(*  *)
	UNIVERSAL_FIXTURE_OPEN				:= 40,	(*  *)
	UNIVERSAL_FIXTURE_CLOSE				:= 50,	(*  *)
	UNIVERSAL_FIXTURE_MEASUREMENT		:= 60,	(*  *)
	UNIVERSAL_FIXTURE_RESET				:= 70,	(*  *)
	UNIVERSAL_FIXTURE_METHOD_DONE		:= 80,
	UNIVERSAL_FIXTURE_EXTENSION			:= 999,	(*  *)
	UNIVERSAL_FIXTURE_ABORTING			:= -10	(*  *)
);
END_TYPE

// ---- DUTs/Libs/Fixtures/UniversalFixture/E_UniversalFixtureStateAbort.TcDUT
{attribute 'strict'}
TYPE E_UniversalFixtureStateAbort :
(
	UNIVERSAL_FIXTURE_ABORT_FILE_LOGGER	:= 0,	(*  *)
	UNIVERSAL_FIXTURE_ABORT_TCP_SERVER	:= 10,	(*  *)
	UNIVERSAL_FIXTURE_ABORT_TCP_CLIENT 	:= 20, 	(*  *)
	UNIVERSAL_FIXTURE_ABORT_DONE		:= 30	(*  *)
);
END_TYPE

// ---- DUTs/Libs/Fixtures/UniversalFixture/E_UniversalFixtureStateInit.TcDUT
{attribute 'strict'}
TYPE E_UniversalFixtureStateInit :
(
	UNIVERSAL_FIXTURE_INIT_TCP_SERVER	:= 0,	(*  *)
	UNIVERSAL_FIXTURE_INIT_TCP_CLIENT	:= 10,	(*  *)
	UNIVERSAL_FIXTURE_INIT_FILE_LOGGER	:= 20,	(*  *)
	UNIVERSAL_FIXTURE_INIT_DONE			:= 30	(*  *)
);
END_TYPE

// ---- DUTs/Libs/Fixtures/UniversalFixture/E_UniversalFixtureStateMeasure.TcDUT
{attribute 'strict'}
TYPE E_UniversalFixtureStateMeasure :
(
	UNIVERSAL_FIXTURE_MEASURE_WAIT_FOR_CLIENT	:= 0,	(* Measurement fixture server is waiting for client connection *)
	UNIVERSAL_FIXTURE_MEASURE_SEND_DATA			:= 10,	(* Measurement fixture server is sending data to measurement device *)
	UNIVERSAL_FIXTURE_MEASURE_RECIVE_DATA		:= 20,	(* Measurement fixture server is waiting for data from measurement device*)
	UNIVERSAL_FIXTURE_MEASURE_DONE				:= 30	(* Measurement sequence finished *)
);
END_TYPE

// ---- DUTs/Libs/Fixtures/UniversalFixture/E_UniversalFixtureStateReset.TcDUT
{attribute 'strict'}
TYPE E_UniversalFixtureStateReset :
(
	UNIVERSAL_FIXTURE_RESETING_FILE_LOGGER				:= 0,	(*  *)
	UNIVERSAL_FIXTURE_RESETING_TCP_SERVER_SHUT_DOWN		:= 10,	(*  *)
	UNIVERSAL_FIXTURE_RESETING_TCP_SERVER_TURN_ON		:= 20,	(*  *)
	UNIVERSAL_FIXTURE_RESETING_TCP_CLIENT_SHUT_DOWN		:= 30,	(*  *)
	UNIVERSAL_FIXTURE_RESETING_TCP_CLIENT_TURN_ON		:= 40,	(*  *)
	UNIVERSAL_FIXTURE_RESETING_DONE						:= 50	(*  *)
);
END_TYPE

// ---- DUTs/Libs/Platform/Common/ST_UniversalPlatform.TcDUT
TYPE ST_UniversalPlatform :
STRUCT
	ref_fbRecipesManager : REFERENCE TO FB_RecipesControler;	(* Main machine recipes controler - provides access to PLC recipes system from HMI *)
	ref_fbAlarmControler : REFERENCE TO FB_AlarmControler; 	(* Main machine alarm controler - provides access to occured errors from HMI*)
END_STRUCT
END_TYPE

// ---- DUTs/Libs/Platform/Universal Machine/E_MachineCtrlState.TcDUT
{attribute 'strict'}
TYPE E_MachineCtrlState :
(
	MACHINE_STATE_UNINITIALIZED 	:= 0,	(*  *)
	MACHINE_STATE_INITIALIZING 		:= 10,	(*  *)
	MACHINE_STATE_READY_INITIALIZED := 20,	(*  *)
	MACHINE_STATE_AUTO				:= 30,	(*  *)
	MACHINE_STATE_AUTO_TO_MANUAL	:= 40,	(*  *)
	MACHINE_STATE_MANUAL			:= 50,	(*  *)
	MACHINE_STATE_MANUAL_TO_AUTO	:= 60,	(*  *)
	MACHINE_STATE_RESET				:= 70,	(*  *)
	MACHINE_STATE_RESET_DONE		:= 80,	(*  *)
	MACHINE_STATE_ABORTING			:= -10,	(*  *)
	MACHINE_STATE_EMERGENCY			:= -20	(*	*)
);
END_TYPE

// ---- DUTs/Libs/Platform/Universal Safety/E_SafetyCtrlState.TcDUT
{attribute 'qualified_only'}
{attribute 'strict'}
TYPE E_SafetyCtrlState :
(
	enum_member := 0
);
END_TYPE

// ---- DUTs/Libs/Platform/Universal Visu/E_VisuCtrlAlarmControlState.TcDUT
{attribute 'strict'}
TYPE E_VisuCtrlAlarmControlState :
(
	VISU_CTRL_ALARM_CONTROLER_WAIT_FOR_CMD 	:= 0,	(*  *)
	VISU_CTRL_ALARM_CONTROLER_INIT			:= 10,	(*  *)
	VISU_CTRL_ALARM_CONTROLER_CLEAR_ALL		:= 20,	(*  *)
	VISU_CTRL_ALARM_CONTTOLER_EXPORT		:= 30,	(*  *)
	VISU_CTRL_ALARM_CONTROLER_ABORT			:= -10	(*  *)
);
END_TYPE

// ---- DUTs/Libs/Platform/Universal Visu/E_VisuCtrlAxisImgType.TcDUT
{attribute 'strict'}
{attribute 'to_string'}
TYPE E_VisuCtrlAxisImgType :
(
	AXIS_TYPE_BECKHOFF_SERVO_AM30XX 	:= 0,	(*  *)
	AXIS_TYPE_BECKHOFF_SERVO_AM80XX 	:= 10,	(*  *)
	AXIS_TYPE_BECKHOFF_SERVO_AM81XX 	:= 20,	(*  *)
	AXIS_TYPE_BECKHOFF_SERVO_AM85XX		:= 30,	(*  *)
	AXIS_TYPE_BECKHOFF_SERVO_AM87XX		:= 40,	(*  *)
	AXIS_TYPE_BECKHOFF_SERVO_AM88XX		:= 50,	(*  *)
	AXIS_TYPE_BECKHOFF_SERVO_AMI812X	:= 60,	(*  *)
	AXIS_TYPE_BECKHOFF_SERVO_AMP80XX	:= 70,	(*  *)
	AXIS_TYPE_BECKHOFF_STEPPER_AG1000 	:= 80,	(*  *)
	AXIS_TYPE_BECKHOFF_STEPPER_AG2250 	:= 90,	(*  *)
	AXIS_TYPE_BECKHOFF_STEPPER_ASXXX 	:= 100,	(*  *)
	AXIS_TYPE_FAULHABER_LM_1257			:= 110,	(*  *)
	AXIS_TYPE_JENNY_SCIENCE_ELAX		:= 120,	(*  *)
	AXIS_TYPE_JENNY_SCIENCE_LINAX_LXC	:= 130,	(*  *)
	AXIS_TYPE_JENNY_SCIENCE_LINAX_LXS	:= 140,	(*  *)
	AXIS_TYPE_JENNY_SCIENCE_LINAX_LXU	:= 150,	(*  *)
	AXIS_TYPE_JENNY_SCIENCE_LINAX_LXE	:= 160,	(*  *)
	AXIS_TYPE_JENNY_SCIENCE_ROTAX_28	:= 170,	(*  *)
	AXIS_TYPE_JENNY_SCIENCE_ROTAX_50	:= 180,	(*  *)
	AXIS_TYPE_JENNY_SCIENCE_ROTAX_110	:= 190,	(*  *)
	AXIS_TYPE_BECKHOFF_XTS_MOVER		:= 200	(*  *)
);
END_TYPE

// ---- DUTs/Libs/Platform/Universal Visu/E_VisuCtrlAxisJogMode.TcDUT
{attribute 'strict'}
TYPE E_VisuCtrlAxisJogMode :
(
	VISU_AXIS_JOG_MODE_STANDARD_SLOW	:= 0,	(*  *)
	VISU_AXIS_JOG_MODE_STANDARD_FAST	:= 1,	(*  *)
	VISU_AXIS_JOG_MODE_CONTINOUS		:= 2,	(*  *)
	VISU_AXIS_JOG_MODE_INCHING			:= 3,	(*  *)
	VISU_AXIS_JOG_MODE_INCHING_MODULO	:= 4	(*  *)
);
END_TYPE

// ---- DUTs/Libs/Platform/Universal Visu/E_VisuCtrlCylinderImgType.TcDUT
{attribute 'strict'}
{attribute 'to_string'}
TYPE E_VisuCtrlCylinderImgType :
(
	CYLINDER_TYPE_SINGLE_COIL := -0,	(*  *)
	CYLINDER_TYPE_DOUBLE_COIL := 10		(*  *)
);
END_TYPE

// ---- DUTs/Libs/Platform/Universal Visu/E_VisuCtrlNavBarState.TcDUT
{attribute 'strict'}
TYPE E_VisuCtrlNavBarState :
(
	NAVIGATION_EMPTY			:= 0,	(*  *)
	NAVIGATION_UNINITIALIZED	:= 1,	(*  *)
	NAVIGATION_INITIALIZING		:= 2,	(*  *)
	NAVIGATION_AUTO 			:= 3,	(*  *)
	NAVIGATION_MANUAL			:= 4,	(*  *)
	NAVIGATION_UTILITIES 		:= 5	(*  *)
);
END_TYPE

// ---- DUTs/Libs/Platform/Universal Visu/E_VisuCtrlPageState.TcDUT
{attribute 'strict'}
TYPE E_VisuCtrlPageState :
(
	SCREEN_UNINITIALIZED 		:= 0,	(*  *)
	SCREEN_INITIALIZING 		:= 1,	(*  *)
	SCREEN_READY_INITIALIZED	:= 2,	(*  *)
	SCREEN_AUTO					:= 3,	(*  *)
	SCREEN_MODE_CHANGE			:= 4,	(*  *)
	SCREEN_MANUAL_CYLINDERS		:= 5,	(*  *)
	SCREEN_MANUAL_MOTORS		:= 6,	(*  *)
	//SCREEN_MANUAL_SAFETY		:= 7,	(*  *)
	SCREEN_MANUAL_INPUTS		:= 7,	(*  *)
	SCREEN_MANUAL_OUTPUTS		:= 8,	(*  *)
	SCREEN_MANUAL_ROBOTS		:= 9,	(*  *)
	SCREEN_MANUAL_OTHERS		:= 10,	(*  *)
	SCREEN_ALARMS				:= 11,	(*  *)
	SCREEN_RECIPES				:= 12,	(*  *)
	SCREEN_RESET				:= 13,	(*  *)
	SCREEN_ABORTING				:= 14,	(*  *)
	SCREEN_EMERGENCY			:= 15	(*  *)
);
END_TYPE

// ---- DUTs/Libs/Platform/Universal Visu/E_VisuCtrlRecipeParameterType.TcDUT
{attribute 'strict'}
TYPE E_VisuCtrlRecipeParameterType :
(
	VISU_CTRL_RECIPES_PARAMETER_TYPE_BOOL 	:= 0,
	VISU_CTRL_RECIPES_PARAMETER_TYPE_INT	:= 1,
	VISU_CTRL_RECIPES_PARAMETER_TYPE_REAL	:= 2,
	VISU_CTRL_RECIPES_PARAMETER_TYPE_STRING := 3
);
END_TYPE

// ---- DUTs/Libs/Platform/Universal Visu/E_VisuCtrlRecipesManagerState.TcDUT
{attribute 'strict'}
TYPE E_VisuCtrlRecipesManagerState :
(
	VISU_CTRL_RECIPE_MANAGER_WAIT_FOR_CMD	:= 0,	(*  *)
	VISU_CTRL_RECIPE_MANAGER_INIT			:= 10,	(*  *)
	VISU_CTRL_RECIPE_MANAGER_CREATE			:= 20,	(*  *)
	VISU_CTRL_RECIPE_MANAGER_LOAD			:= 30,	(*  *)
	VISU_CTRL_RECIPE_MANAGER_READ			:= 40,	(*  *)
	VISU_CTRL_RECIPE_MANAGER_RELOAD			:= 50,	(*  *)
	VISU_CTRL_RECIPE_MANAGER_BACKUP			:= 60,	(*  *)
	VISU_CTRL_RECIPE_MANAGER_RESTORE		:= 70,	(*  *)
	VISU_CTRL_RECIPE_MANAGER_REMOVE			:= 80,	(*  *)
	VISU_CTRL_RECIPE_MANAGER_RELOAD_EXT		:= 90,
	VISU_CTRL_RECIPE_MANAGER_ABORT 			:= -10	(*  *)
);
END_TYPE

// ---- DUTs/Libs/Platform/Universal Visu/E_VisuCtrlRobotImgType.TcDUT
{attribute 'strict'}
{attribute 'to_string'}
TYPE E_VisuCtrlRobotImgType :
(
	ROBOT_TYPE_MITSUBISHI_6_AXIS 	:= 0,	(*  *)
	ROBOT_TYPE_MITSUBISHI_SCARA 	:= 10	(*  *)
);
END_TYPE

// ---- DUTs/Libs/Platform/Universal Visu/E_VisuCtrlSingleAxisState.TcDUT
{attribute 'strict'}
TYPE E_VisuCtrlSingleAxisState :
(
	VISU_CTRL_AXIS_WAIT_FOR_CMD := 0,	(* *)
	VISU_CTRL_AXIS_INIT			:= 10,	(*  *)
	VISU_CTRL_AXIS_RESET		:= 20,	(*  *)
	VISU_CTRL_AXIS_HOME			:= 30,	(*  *)
	VISU_CTRL_AXIS_HALT			:= 40,	(*  *)
	VISU_CTRL_AXIS_JOG_POSITIVE	:= 50,	(*  *)
	VISU_CTRL_AXIS_JOG_NEGATIVE	:= 60,	(*  *)
	VISU_CTRL_AXIS_ABORT		:= -10	(*  *)
);
END_TYPE

// ---- DUTs/Libs/Platform/Universal Visu/E_VisuCtrlSingleCylinderState.TcDUT
{attribute 'strict'}
TYPE E_VisuCtrlSingleCylinderState :
(
	VISU_CTRL_CYLINDER_WAIT_FOR_CMD := 0,	(*  *)
	VISU_CTRL_CYLINDER_INIT			:= 10,	(*  *)
	VISU_CTRL_CYLINDER_RESET		:= 20,	(*  *)
	VISU_CTRL_CYLINDER_GO_HOME		:= 30,	(*  *)
	VISU_CTRL_CYLINDER_GO_ACTIVE	:= 40,	(*  *)
	VISU_CTRL_CYLINDER_GO_RELEASE	:= 50,	(*  *)
	VISU_CTRL_CYLINDER_ABORT		:= -10	(*  *)
);
END_TYPE

// ---- DUTs/Libs/Platform/Universal Visu/E_VisuCtrlSingleRobotState.TcDUT
{attribute 'strict'}
TYPE E_VisuCtrlSingleRobotState :
(
	VISU_CTRL_ROBOT_WAIT_FOR_CMD	 := 0,	(*  *)
	VISU_CTRL_ROBOT_INIT			:= 10,	(*  *)
	VISU_CTRL_ROBOT_ERR_RESET		:= 20,	(*  *)
	VISU_CTRL_ROBOT_CONTROLLER_RESET:= 30,	(*  *)
	VISU_CTRL_ROBOT_GO_HOME			:= 40,	(*  *)
	VISU_CTRL_ROBOT_DO_ACTION		:= 50,	(*  *)
	VISU_CTRL_ROBOT_GO_AUTO			:= 60,	(*  *)
	VISU_CTRL_ROBOT_UPDATE_RECIPES	:= 70,	(*  *)
	VISU_CTRL_ROBOT_CYCLE_PAUSE		:= 80,	(*  *)
	VISU_CTRL_ROBOT_CYCLE_STOP		:= 90,	(*  *)
	VISU_CTRL_ROBOT_RESTORE_CYCLE	:= 100,	(*  *)
	VISU_CTRL_ROBOT_RESTORE_AUTO	:= 110,	(*  *)
	VISU_CTRL_ROBOT_BATTERY_RESET	:= 120,	(*  *)	
	VISU_CTRL_ROBOT_ABORT			:= -10	(*  *)
);
END_TYPE

// ---- DUTs/Libs/Platform/Universal Visu/E_VisuCtrUniversalMachineState.TcDUT
{attribute 'strict'}
TYPE E_VisuCtrUniversalMachineState :
(	
	VISU_CTRL_UNIVERSAL_MACHINE_WAIT_FOR_CMD	 	:= 0,	(*  *)
	VISU_CTRL_UNIVERSAL_MACHINE_INIT				:= 10,	(*  *)
	VISU_CTRL_UNIVERSAL_MACHINE_RESET				:= 20,	(*  *)
	VISU_CTRL_UNIVERSAL_MACHINE_START_AUTO			:= 30,	(*  *)
	VISU_CTRL_UNIVERSAL_MACHINE_STOP_AUTO			:= 40,	(*  *)
	VISU_CTRL_UNIVERSAL_MACHINE_SWITCH_TO_MANUAL	:= 50,	(*  *)
	VISU_CTRL_UNIVERSAL_MACHINE_SWITCH_TO_AUTO		:= 60,	(*  *)
	VISU_CTRL_UNIVERSAL_MACHINE_ABORT				:= -10	(*  *)
);
END_TYPE

// ---- DUTs/Libs/Platform/Universal Visu/ST_VisuCtrlAxisFrame.TcDUT
TYPE ST_VisuCtrlAxisFrame EXTENDS ST_VisuCtrlUnitFrame :
STRUCT
	sUnit 				: STRING := 'Unknown';	(*  *)
	
	btnInit 			: BOOL;						(*  *)
	btnAbort 			: BOOL;						(*  *)
	btnReset			: BOOL;						(*  *)
	btnHome 			: BOOL;						(*  *)
	btnHalt				: BOOL;						(*  *)
	btnJogPositive 		: BOOL;						(*  *)
	btnJogNegative 		: BOOL;						(*  *)
	
	bActive				: BOOL;						(*  *)
	bHomed 				: BOOL;						(*  *)
	bInPosition 		: BOOL;						(*  *)
	bHalted				: BOOL;						(*  *)
	bError				: BOOL;						(*  *)
	iErrorID			: UDINT;					(*  *)
	
	lrActualPosition	: LREAL;					(*  *)
	lrActualVelocity	: LREAL;					(*  *)
	lrLagError			: LREAL;					(*  *)
	
	lrSetPosition		: LREAL;					(*  *)
	lrSetVelocity		: LREAL;					(*  *)
	
	lrOverride			: LREAL := 30.0;			(*  *)
	
	lrJogDistance 		: LREAL;					(*  *)
	lrJogVelocity		: LREAL;					(*  *)
	lrJogAcceleration	: LREAL;					(*  *)
	lrJogDeceleartion	: LREAL;					(*  *)
	
	sAxisImage			: STRING;					(*  *)
	eJogMode			: E_VisuCtrlAxisJogMode;	(*  *)
	eAxisState			: E_AxisState;				(*  *)
END_STRUCT
END_TYPE

// ---- DUTs/Libs/Platform/Universal Visu/ST_VisuCtrlCylinderFrame.TcDUT
TYPE ST_VisuCtrlCylinderFrame EXTENDS ST_VisuCtrlUnitFrame :
STRUCT
	btnInit				: BOOL;				(*  *)
	btnAbort			: BOOL;				(*  *)
	btnReset			: BOOL;				(*  *)
	btnGoHome 			: BOOL;				(*  *)
	btnGoActive 		: BOOL;				(*  *)
	btnRealase 			: BOOL;				(*  *)
	
	bSensorHome 		: BOOL;				(*  *)
	bSensorActive 		: BOOL;				(*  *)
	bPositionHold		: BOOL;				(*  *)
	bError				: BOOL;				(*  *)
	iErrorID			: UDINT;			(*  *)
	
	tActiveMovement 	: TIME;				(*  *)
	tHomeMovement 		: TIME;				(*  *)
	
	sActiveDescription 	: STRING;			(*  *)
	sHomeDescription 	: STRING;			(*  *)
	sStateDescription	: STRING;			(*  *)
	
	sCylinderImage		: STRING;			(*  *)
	eCylinderState		: E_CylinderState;	(*  *)
END_STRUCT
END_TYPE

// ---- DUTs/Libs/Platform/Universal Visu/ST_VisuCtrlFixtureFrame.TcDUT
TYPE ST_VisuCtrlFixtureFrame EXTENDS ST_VisuCtrlUnitFrame:
STRUCT
END_STRUCT
END_TYPE

// ---- DUTs/Libs/Platform/Universal Visu/ST_VisuCtrlInputFrame.TcDUT
TYPE ST_VisuCtrlInputFrame EXTENDS ST_VisuCtrlUnitFrame:
STRUCT
	bIn				: BOOL;								(*  *)
	bForceIn		: BOOL;								(*  *)
	bForceDisabled	: BOOL	:=TRUE ;					(*  *)
	sModuleType		: STRING;							(* Module type e.g. EL1xxx *)
	sPortID			: STRING;							(* Wire id connected to port *)
END_STRUCT
END_TYPE

// ---- DUTs/Libs/Platform/Universal Visu/ST_VisuCtrlOutputFrame.TcDUT
TYPE ST_VisuCtrlOutputFrame EXTENDS ST_VisuCtrlUnitFrame :
STRUCT
	btnOut 			: BOOL; 		(* This button allows to control ouptu manualy if it's set as controlable *)
	bOut 			: BOOL;			(* This bit indicates the status of output in manual mode *)
	bControlable	: BOOL;			(* This bit is used to lock control of output via manual mode - read access only *)
	sModuleType		: STRING;		(* Module type e.g. EL1xxx *)
	sPortID			: STRING;		(* Wire id connected to port *)
END_STRUCT
END_TYPE

// ---- DUTs/Libs/Platform/Universal Visu/ST_VisuCtrlRecipeParameter.TcDUT
TYPE ST_VisuCtrlRecipeParameter :
STRUCT
	bValue		: REFERENCE TO BOOL;	(* Reference to bit value of recipe parameter *)
	iValue		: REFERENCE TO DINT;	(* Reference to integer value of recipe parameter *)
	rValue		: REFERENCE TO REAL;	(* Reference to real value of recipe parameter *)
	sValue		: REFERENCE TO STRING;	(* Reference to string value of recipe parameter *)
	sName 		: REFERENCE TO STRING;	(* Reference to name of recipe parameter *)
	sFileValue	: REFERENCE TO STRING;	(* Reference to bit value of recipe parameter *)
END_STRUCT
END_TYPE

// ---- DUTs/Libs/Platform/Universal Visu/ST_VisuCtrlRecipesManager.TcDUT
TYPE ST_VisuCtrlRecipesManager :
STRUCT
	btnCreate				: BOOL;																						(*  *)
	btnRemove				: BOOL;																						(*  *)
	btnLoad					: BOOL;																						(* Load recipe button for HMI frame *)
	btnRead					: BOOL;																						(* Read recipe button for HMI frame *)
	btnReaload 				: BOOL;																						(* Reload recipes button for HMI frame *)
	btnBackup				: BOOL;																						(* Backup recipes to external directory button for HMI freame*)
	btnRestore				: BOOL;																						(* Restore recipes from external directory button for HMI frame *)
	bError					: BOOL;																						(* Error occured while executing last command *)
	eRecipesManagerReturns	: E_RecipesManagerReturns;																	(* Result of last executed command *)
	eReacipeManagerState	: E_RecipesManagerState;																	(* Current state of Recipe Manager *)
	sRecipeName				: STRING;																					(* Current selected recipe name *)
	iSelectedRecipe			: USINT;
	//arrRecipeNames			: ARRAY	[0..iMAX_NUMBER_OF_VARIABLES_IN_RECIPES - 1] OF STRING(iMAX_RECIPE_NAME_LENGTH);(* Array of recipes detected at demanded directory *)
	arrRecipeNames			: ARRAY	[0..127] OF STRING;																	(* Array of recipes names detected at demanded directory *)
	sRecipeDescription		: STRING(iMAX_RECIPE_DESCRIPTION_LENGTH); 													(* Description of selected recipe *)
	sRestoreBackupPath		: STRING(iMAX_RECIPE_RESTOR_BACKUP_PATH_LENGTH);											(* Path for backup/restoring of recipes *)
END_STRUCT
END_TYPE

// ---- DUTs/Libs/Platform/Universal Visu/ST_VisuCtrlRobotFrame.TcDUT
TYPE ST_VisuCtrlRobotFrame EXTENDS ST_VisuCtrlUnitFrame :
STRUCT
	btnInit						: BOOL;				(*  *)
	btnAbort					: BOOL;				(*  *)
	btnErrorReset				: BOOL;				(*  *)
	btnControllerReset			: BOOL;				(*  *)
	btnBatteryReset				: BOOL;				(*  *)
	btnGoHome 					: BOOL;				(*  *)
	btnDoAction	 				: BOOL;				(*  *)
	btnUpdateRecipes			: BOOL;				(*  *)
	btnGoAuto 					: BOOL;				(*  *)
	btnCyclePause				: BOOL;				(*  *)
	btnCycleStop				: BOOL;				(*  *)
	btnRestoreCycle 			: BOOL;				(*  *)
	btnRestoreAuto	 			: BOOL;				(*  *)
	btnModeSwitch	 			: BOOL;				(*  *)

	bError						: BOOL;				(*  *)
	bInit						: BOOL;	
	bPowerOn					: BOOL;	
	bBatteryLow					: BOOL;	
	bIsHomed					: BOOL;
	bServoOn					: BOOL;				(*  *)
	bServoOff 					: BOOL;
	bStarted					: BOOL;
	bStopped					: BOOL;				(*  *)
	bPaused						: BOOL;
	bUninitialized				: BOOL;
	bDoAction					: BOOL;
	bAutoButtonDisable			: BOOL;	
	bActionButtonDisable		: BOOL;	
	bHomeButtonDisable 			: BOOL;
	bPausingButtonDisable 		: BOOL;
	bRestoreCycleButtonDisable  : BOOL;
	bStoppingButtonDisable	    : BOOL;
	bRestoreAutoButtonDisable   : BOOL;
	bInitButtonDisable			: BOOL;
	bModeSwitchState			: BOOL;
	bModeSwitchButtonDisabled 	: BOOL;
	
	sErrorDescription			: STRING;			(*  *)
	iActionNumber				: UINT := 51;		(*  *)
	iOverride					: USINT := 100;
	sStateDescription			: STRING;			(*  *)
	
	sRobotImage					: STRING;			(*  *)
	eRobotState					: E_CR800State;		(*  *)
END_STRUCT
END_TYPE

// ---- DUTs/Libs/Platform/Universal Visu/ST_VisuCtrlUnitFrame.TcDUT
TYPE ST_VisuCtrlUnitFrame :
STRUCT
	sName : STRING := 'Unknown';	(* Name of object for any visu frame *)
END_STRUCT
END_TYPE

// ---- DUTs/Libs/Robots/Mitsubishi/CR800/EtherCAT Registers/ST_CR800EthercatData.TcDUT
(* Enum for data handling beetwen PLC and CR800. Used in FB_CR800Ethercat *) 
TYPE ST_CR800EthercatData :
STRUCT

	arrRegistersInput 			AT%I* 	: ARRAY[6000..6127] OF INT ; 		(*Input process data (RWr)*)
	arrSignalsInputRaw			AT%I*	: ARRAY[0..31]		OF BYTE ; 		(*Input process data (RX) before convertion to easier to use. 
																			  This data are is used only in MR_ConvertEthercatData*)
	arrSignalsInputConverted			: ARRAY[6000..6255]	OF BOOL ; 		(*Input process data (RX) after convertion to esier to uses. 
																			  This data are used in program*)
	
	arrRegistersOutput 			AT%Q* 	: ARRAY[6000..6127] OF INT ; 		(*Output process data (RWr)*)
	arrSignalsOutputRaw			AT%Q*	: ARRAY[0..31] 		OF BYTE ; 		(*Output process data (RX) before convertion to easier to use. 
																			  This data are is used only in MR_ConvertEthercatData*)
	arrSignalsOutputConverted			: ARRAY[6000..6255] OF BOOL ; 		(*Output process data (RX) after convertion to esier to uses. 
																			  This data are used in program*)

	iInfoDataState				AT%I* 	: INT ;								(* Indicates status of ethercat communication *)
	
END_STRUCT
END_TYPE

// ---- DUTs/Libs/Robots/Mitsubishi/CR800/E_CR800Error.TcDUT
(* Enum for error handling FB_CR800Ethercat *)
{attribute 'strict'}
{attribute 'to_string'}
TYPE E_CR800Error :
(
	CR800_ERROR_OK										:= 0,	(*  *)
	CR800_ERROR_ETHERCAT_CHECK_FAIL						:= 5,	(*  *) 
	CR800_ERROR_POWER_CHECK_FAIL						:= 10,	(*  *) 
	CR800_ERROR_EMERGENCY_STOP_OCCURING					:= 20, 	(*  *)
	CR800_ERROR_AUTO_MODE_CHECK_FAIL					:= 30,	(*  *)
	CR800_ERROR_GRANTING_OPERATION_RIGHTS_TIMED_OUT 	:= 40,	(*  *)
	CR800_ERROR_ABORTING_OPERATION_RIGHTS_TIMED_OUT 	:= 50,	(*  *)
	CR800_ERROR_SERVO_ON_TIMED_OUT						:= 60,	(*  *)
	CR800_ERROR_CANT_RESET_PRG_DURING_PRG_RUN			:= 70,	(*  *)
	CR800_ERROR_RESET_PRG_TIMED_OUT						:= 80,	(*  *)
	CR800_ERROR_START_PRG_TIMED_OUT						:= 90,	(*  *)
	CR800_ERROR_SEND_COMMAND_TIMED_OUT					:= 100,	(*  *)	
	CR800_ERROR_RECEIVE_COMMAND_TIMED_OUT				:= 110,	(*  *)	
	CR800_ERROR_CANT_GO_AUTO_WITHOUT_BEEING_HOMED		:= 120,	(*  *)		
	CR800_ERROR_CANT_DO_ACTION_WITHOUT_BEEING_AUTO		:= 130,	(*  *)	
	CR800_ERROR_CANT_DO_SYSTEM_ACTION_IN_THIS_REQUEST	:= 140,	(*  *)
	CR800_ERROR_CR800_ERROR_OCCURING					:= 150	(*  *) 
		
);
END_TYPE

// ---- DUTs/Libs/Robots/Mitsubishi/CR800/StateMachine/E_CR800State.TcDUT
{attribute 'strict'}
TYPE E_CR800State :
(
	CR800_UNINITIALIZED				:= 0,	(* Cr800 is uninitialized *)
	CR800_INITIALIZING				:= 10,	(* Initialization in a progress *)
	CR800_READY_INITIALIZED			:= 20,	(*  *)
	CR800_IDLE_NOT_HOMED			:= 30,	(* Cr800 ready to work *)

	CR800_GOING_HOME				:= 40,	(* Cr800 is going to a home position *)
	CR800_GOING_HOME_DONE			:= 50,	(* Cr800 is in a home position *)
	CR800_IDLE_HOMED				:= 60,	(* Cr800 is ready for requests and homed *)
	CR800_UPDATING_RECIPIES			:= 70,	(* Cr800 is updating recipies*)
	CR800_UPDATE_RECIPIES_DONE		:= 80,	(* Cr800 updated the repcies*)

	CR800_GOING_AUTO				:= 100,	(* CR800 is going to the auto mode *)
	CR800_GOING_AUTO_DONE			:= 110,	(* CR800 is in the auto mode *)
	CR800_IDLE_AUTO					:= 120, (* CR800 is ready to operate in auto mode*)
	CR800_DOING_ACTION				:= 130,	(* Do action*)
	CR800_DOING_ACTION_DONE			:= 140,	(* Done - action *)

	CR800_CYCLE_STOPPING			:= 200,	(* Cr800 program stops after the cycle is finished *)	
	CR800_CYCLE_STOPING_DONE		:= 210,	(* Cr800 program stops after the cycle is finished done *)	
	CR800_IDLE_AUTO_PAUSED			:= 220,	(* CR800 paused and program is off *)
	CR800_AUTO_RESTORING			:= 230, (* CR800 is going to restore the auto mode *)
	CR800_AUTO_RESTORING_DONE		:= 240, (* CR800 restored the auto mode *)
	
	CR800_CYCLE_PAUSING				:= 300,	(* Cr800 program is going to stop immediately and pause *)	
	CR800_CYCLE_PAUSING_DONE		:= 310,	(* Cr800 program is going to stop immediately and pause done *)	
	CR800_IDLE_CYCLE_PAUSED			:= 320,	(* CR800 program is paused *)
	CR800_CYCLE_RESTORING			:= 330, (* CR800 is going to restore the cycle mode *)
	CR800_CYCLE_RESTORING_DONE		:= 340, (* CR800 restored the cycle *)
	
	CR800_SEND_POSITION_1			:= 400,
	CR800_SEND_POSITION_1_DONE		:= 410,
	CR800_SEND_POSITION_2			:= 420,
	CR800_SEND_POSITION_2_DONE		:= 430,
	CR800_GET_POSITION				:= 440,
	CR800_GET_POSITION_DONE			:= 450,
	
	CR800_RESET						:= 500,	(* Reseting the function block *)
	CR800_RESET_DONE				:= 510,	(* Reset done *)
	
	CR800_IN_EXTERNAL_ERROR			:= -10,	(* FB is in an extrnal error *)
	
	CR800_ABORTING 					:= -20	(* Aborting *)
	
);
END_TYPE

// ---- DUTs/Libs/Robots/Mitsubishi/CR800/StateMachine/E_CR800StateAborting.TcDUT
{attribute 'strict'}
TYPE E_CR800StateAborting :
(
	CR800_ABORTING_IDLE				:= 0,	(* DUMMY *)
	CR800_ABORTING_ENABLE_RIGHTS	:= 5,	(* Enable rights *)
	CR800_ABORTING_PRGM_STOP		:= 10,	(* Pogram stop *)
	CR800_ABORTING_PRGM_RESET		:= 20,	(* Program reset *)
	CR800_ABORTING_SERVO_OFF		:= 30,	(* Servo off *)
	CR800_ABORTING_DONE				:= 40	(* Aborting done *)	
); 
END_TYPE

// ---- DUTs/Libs/Robots/Mitsubishi/CR800/StateMachine/E_CR800StateCommandExchange.TcDUT
(* Enum for exchange the data in FB_CR800Ethercat *)
{attribute 'strict'}
TYPE E_CR800StateCommandExchange :
(
	CR800_CMD_EXCHANGE_IDLE							:= 0,	(*  *)
	CR800_CMD_EXCHANGE_SEND_DATA	 				:= 10,	(*  *)
	CR800_CMD_EXCHANGE_WAIT_FOR_DATA				:= 15,	(*  *)
	CR800_CMD_EXCHANGE_WAIT_FOR_CONFIRMATION 		:= 20,	(*  *)
	CR800_CMD_EXCHANGE_SEND_CONFIRMATION			:= 25,	(*  *)
	CR800_CMD_EXCHANGE_RESET_ITERLOCKS				:= 30,	(*  *)
	CR800_CMD_EXCHANGE_WAIT_FOR_RESET_COMMAND		:= 35,	(*  *)
	CR800_CMD_EXCHANGE_WAIT_FOR_RESET_CONFIRMATION	:= 40,	(*  *)
	CR800_CMD_EXCHANGE_SEND_RESET_CONFIRMATION		:= 45,	(*  *)
	CR800_CMD_EXCHANGE_DONE							:= 50	(*  *)
);
END_TYPE

// ---- DUTs/Libs/Robots/Mitsubishi/CR800/StateMachine/E_CR800StateCyclePausing.TcDUT
{attribute 'strict'}
TYPE E_CR800StateCyclePausing :
(
	CR800_CYCLE_PAUSING_IDLE	:= 0,	(* DUMMY *)
	CR800_CYCLE_PAUSING			:= 10,	(* Pausing in opearation *)
	CR800_CYCLE_PAUSING_DONE	:= 30	(* Pausing done *)
); 
END_TYPE

// ---- DUTs/Libs/Robots/Mitsubishi/CR800/StateMachine/E_CR800StateCycleStopping.TcDUT
{attribute 'strict'}
TYPE E_CR800StateCycleStopping :
(
	CR800_CYCLE_STOPPPING_IDLE				:= 0,	(* DUMMY *)
	CR800_CYCLE_STOPPPING_SEND_REQUEST		:= 10,	(* Send "STOP CYCLE" reqest *)
	CR800_CYCLE_STOPPPING_WAIT_FOR_STOP		:= 20,	(* Wait for information that "STOP CYCLE" mode is done *)
	CR800_CYCLE_STOPPPING_RESET_VARIABLES	:= 30,	(* Wait for information that "STOP CYCLE" mode is done *)
	CR800_CYCLE_STOPPPING_DONE				:= 40	(* Action done *)
); 
END_TYPE

// ---- DUTs/Libs/Robots/Mitsubishi/CR800/StateMachine/E_CR800StateDoingRequest.TcDUT
{attribute 'strict'}
TYPE E_CR800StateDoingRequest :
(
	CR800_DOING_REQUEST_IDLE					:= 0,	(* DUMMY *)
	CR800_DOING_REQUEST_SEND_REQUEST			:= 10,	(* Send order reqest *)
	CR800_DOING_REQUEST_WAIT_FOR_CONFIRM		:= 20,	(* Wait for information that order is done *)
	CR800_DOING_REQUEST_DONE					:= 30	(* Request done *)
); 
END_TYPE

// ---- DUTs/Libs/Robots/Mitsubishi/CR800/StateMachine/E_CR800StateHoming.TcDUT
{attribute 'strict'}
TYPE E_CR800StateHoming :
(
	CR800_HOMING_IDLE					:= 0,	(* DUMMY *)
	CR800_HOMING_RESET_PROGRAM			:= 10,	(* Reset the program *)
	CR800_HOMING_RESET_CYCLE_VARIABLES	:= 20,	(* Reset variables from doing action *)
	CR800_HOMING_START_PROGRAM			:= 30,	(* Start the program *)
	CR800_HOMING_SEND_REQUEST			:= 40,	(* Send homing reqest *)
	CR800_HOMING_WAIT_FOR_HOME			:= 50,	(* Wait for information that homing is done *)
	CR800_HOMING_DONE					:= 60	(* Homing done *)
); 
END_TYPE

// ---- DUTs/Libs/Robots/Mitsubishi/CR800/StateMachine/E_CR800StateInitializing.TcDUT
{attribute 'strict'}
TYPE E_CR800StateInitializing :
(
	CR800_INIT_IDLE								:= 0,	(* DUMMY *)
	CR800_INIT_ETHERCAT_CHCEK					:= 5,	(* Check for ethercat *)
	CR800_INIT_POWER_CHCECK						:= 10,	(* Check for power *)
	CR800_INIT_EMERG_STOP_CHCECK				:= 20,	(* Check for emergency stop *)
	CR800_INIT_CHECK_FOR_AUTO_MODE				:= 30,	(* Check for remote mode *)
	CR800_INIT_ENABLE_RIGHTS					:= 40,	(* Enable operation rights *)
	CR800_INIT_SERVO_ON							:= 50,	(* Servo on *)
	CR800_INIT_PROGRAM_RESET					:= 60,	(* Reset program *)
	CR800_INIT_PROGRAM_START					:= 70,	(* Start the program *)	
	CR800_INIT_SET_INITIAL_PARAMETERS_REQUEST 	:= 80,	(* Send set initial parameters request*)
	CR800_INIT_ROBOT_FIRST_CYCLE_DONE			:= 90,	(* Wait for information that first cycle is done *)
	CR800_INIT_DONE								:= 100	(* Initalization done *)
); 
END_TYPE

// ---- DUTs/Libs/Robots/Mitsubishi/CR800/StateMachine/E_CR800StateSendPosition.TcDUT
{attribute 'strict'}
TYPE E_CR800StateSendPosition :
(
	CR800_SEND_POSITION_CONVERTING				:= 0,	(* DUMMY *)
	CR800_SEND_POSITION_SENDING					:= 10
); 
END_TYPE

// ---- DUTs/Libs/Robots/Mitsubishi/CR800/ST_CR800UserDefinedArea.TcDUT
(* Enum for data handling beetwen PLC and CR800. Used in FB_CR800Ethercat *) 
TYPE ST_CR800UserDefinedArea :
STRUCT
	bArea1 		: BOOL;
	bArea2 		: BOOL;
	bArea3 		: BOOL;
	bArea4 		: BOOL;
	bArea5 		: BOOL;
	bArea6 		: BOOL;
	bArea7 		: BOOL;
	bArea8 		: BOOL;	
END_STRUCT
END_TYPE

// ---- DUTs/Libs/Robots/Mitsubishi/E_RobotActions.TcDUT
{attribute 'qualified_only'}
{attribute 'strict'}
TYPE E_RobotActions :
(
	(*System actions - DO NOT USE*)
		FIRST_CYCLE := 0, (*RESERVED - DO NOT USE (used in separated method MR_Init*)
		DO_HOMING 	:= 1, (*RESERVED - DO NOT USE (used in separated method MR_GoHome*)
	
	(*HOMED ACTIONS - from 11 to 50 (actions that a robot can do while is in home position)*)
		GO_AUTO			:= 11, (*RESERVED - DO NOT USE (used in separated method MR_GoAuto*)
		UPDATE_RECIPIES	:= 12, (*RESERVED - DO NOT USE (used in separated method MR_UpdateRecipies*)
		(*
		HOMED_ACTION03	:= 13,
		.
		. etc. 
		HOMED_ACTION50	:= 50,
		*)
	
	(*AUTO ACTIONS - from 51 to 100 (actions that a robot can do while is in auto mode)*)
		PICK_AND_PLACE	:= 51, (* EXAMPLE *)
		DO_CIRCLE		:= 52 (* EXAMPLE *)
		(*AUTO_ACTION03	:= 53,
	  	.
		.
		. etc.
		AUTO_ACTION50	:= 100
		*)
)UINT;
END_TYPE

// ---- DUTs/Libs/Robots/Mitsubishi/E_RobotSystemActions.TcDUT
(* Enums for setting proper action in proper request. Used only internaly for FB_CR800Ethercat *) 
//{attribute 'qualified_only'}
//{attribute 'strict'}
TYPE E_RobotSystemActions :
(
	SET_INITIAL_PARAMETERS 	:= 0, 
	DO_HOMING 				:= 1,
	GO_AUTO					:= 11,
	UPDATE_RECIPIES 		:= 12	
)UINT;
END_TYPE

// ---- DUTs/Libs/Utilities/CSV Data Exchanger/E_CSVDataExchangerCountColumnsState.TcDUT
{attribute 'strict'}
TYPE E_CSVDataExchangerCountColumnsState :
(
	CSV_DATA_EXCHANGER_COUNT_COLUMNS_OPEN_FILE 				:= 0,
	CSV_DATA_EXCHANGER_COUNT_COLUMNS_WAIT_FOR_OPENING		:= 10,	
	CSV_DATA_EXCHANGER_COUNT_COLUMNS_READ_SINGLE_LINE 		:= 20,	
	CSV_DATA_EXCHANGER_COUNT_COLUMNS_WAIT_FOR_READING		:= 30,	
	CSV_DATA_EXCHANGER_COUNT_COLUMNS_COUNT					:= 40,	
	CSV_DATA_EXCHANGER_COUNT_COLUMNS_CLOSE_FILE				:= 50,	
	CSV_DATA_EXCHANGER_COUNT_COLUMNS_WAIT_FOR_CLOSING		:= 60,
	CSV_DATA_EXCHANGER_COUNT_COLUMNS_READING_DONE			:= 70
);
END_TYPE

// ---- DUTs/Libs/Utilities/CSV Data Exchanger/E_CSVDataExchangerInitState.TcDUT
{attribute 'strict'}
TYPE E_CSVDataExchangerInitState :
(
	CSV_DATA_EXCHANGER_INIT_CREATE_DIR		:= 0,	(* Getting current time *)
	CSV_DATA_EXCHANGER_INIT_GET_TIME 		:= 10,	(* Creating directory if doesn't exist *)
	CSV_DATA_EXCHANGER_INIT_CREATE_FILE		:= 20,	(* Creating empty file of logger *)
	CSV_DATA_EXCHANGER_INIT_ADD_HEADER		:= 30,	(* Adding header at the beggining of file *)
	CSV_DATA_EXCHANGER_INIT_CLOSE_FILE		:= 40,	(* Closing file *)
	CSV_DATA_EXCHANGER_INIT_DONE 			:= 50	(* Initiazlization done *)
);
END_TYPE

// ---- DUTs/Libs/Utilities/CSV Data Exchanger/E_CSVDataExchangerInsertIntoTableState.TcDUT
{attribute 'strict'}
TYPE E_CSVDataExchangerInsertIntoTableState :
(
	CSV_DATA_EXCHANGER_INSERT_INTO_TABLE_OPEN_FILE 							:= 0,
	CSV_DATA_EXCHANGER_INSERT_INTO_TABLE_WAIT_FOR_OPENING					:= 10,	
	CSV_DATA_EXCHANGER_INSERT_INTO_TABLE_CONV_ONE_RECORD_TO_CSV 			:= 20,	
	CSV_DATA_EXCHANGER_INSERT_INTO_TABLE_WRITE_SINGLE_LINE					:= 30,	
	CSV_DATA_EXCHANGER_INSERT_INTO_TABLE_WAIT_FOR_WRITTING_SINGLE_LINE		:= 40,	
	CSV_DATA_EXCHANGER_INSERT_INTO_TABLE_CLOSE_FILE							:= 50,	
	CSV_DATA_EXCHANGER_INSERT_INTO_TABLE_WAIT_FOR_CLOSING					:= 60,
	CSV_DATA_EXCHANGER_INSERT_INTO_TABLE_WRITTING_DONE						:= 70
);
END_TYPE

// ---- DUTs/Libs/Utilities/CSV Data Exchanger/E_CSVDataExchangerSelectAllState.TcDUT
{attribute 'strict'}
TYPE E_CSVDataExchangerSelectAllState :
(
	CSV_DATA_EXCHANGER_SELECT_ALL_OPEN_FILE 			:= 0,
	CSV_DATA_EXCHANGER_SELECT_ALL_WAIT_FOR_OPENING		:= 10,	
	CSV_DATA_EXCHANGER_SELECT_ALL_READ_SINGLE_LINE 		:= 20,	
	CSV_DATA_EXCHANGER_SELECT_ALL_WAIT_FOR_READING		:= 30,	
	CSV_DATA_EXCHANGER_SELECT_ALL_PARSE_SINGLE_LINE		:= 40,	
	CSV_DATA_EXCHANGER_SELECT_ALL_CLOSE_FILE			:= 50,	
	CSV_DATA_EXCHANGER_SELECT_ALL_WAIT_FOR_CLOSING		:= 60,
	CSV_DATA_EXCHANGER_SELECT_ALL_READING_DONE			:= 70
);
END_TYPE

// ---- DUTs/Libs/Utilities/CSV Data Exchanger/E_CSVDataExchangerSelectRowState.TcDUT
{attribute 'strict'}
TYPE E_CSVDataExchangerSelectRowState :
(
	CSV_DATA_EXCHANGER_SELECT_ROW_OPEN_FILE 			:= 0,
	CSV_DATA_EXCHANGER_SELECT_ROW_WAIT_FOR_OPENING		:= 10,	
	CSV_DATA_EXCHANGER_SELECT_ROW_READ_SINGLE_LINE 		:= 20,	
	CSV_DATA_EXCHANGER_SELECT_ROW_WAIT_FOR_READING		:= 30,	
	CSV_DATA_EXCHANGER_SELECT_ROW_PARSE_SINGLE_LINE		:= 40,	
	CSV_DATA_EXCHANGER_SELECT_ROW_CLOSE_FILE			:= 50,	
	CSV_DATA_EXCHANGER_SELECT_ROW_WAIT_FOR_CLOSING		:= 60,
	CSV_DATA_EXCHANGER_SELECT_ROW_READING_DONE			:= 70
);
END_TYPE

// ---- DUTs/Libs/Utilities/CSV Data Exchanger/E_CSVDataExchangerSetNewPathState.TcDUT
{attribute 'strict'}
TYPE E_CSVDataExchangerSetNewPathState :
(
	CSV_DATA_EXCHANGER_SET_NEW_PATH_CHANGE_PATH			:= 0,
	CSV_DATA_EXCHANGER_SET_NEW_PATH_COUNT_FILE_COLUMNS	:= 10
);
END_TYPE

// ---- DUTs/Libs/Utilities/CSV Data Exchanger/E_CSVDataExchangerState.TcDUT
{attribute 'strict'}
TYPE E_CSVDataExchangerState :
(
	CSV_DATA_EXCHANGER_UNINITIALIZED 				:= 0,	(* Not ready to work *)
	CSV_DATA_EXCHANGER_INITIALIZING					:= 10,	(* Preparing to work *)
	CSV_DATA_EXCHANGER_READY 						:= 20,	(* Ready to work *)
	CSV_DATA_EXCHANGER_IDLE				 			:= 30,	(* Ready to work, waiting for logs in buffer *)
	CSV_DATA_EXCHANGER_SELECT_ALL					:= 40,	
	CSV_DATA_EXCHANGER_SELECT_ROW					:= 50,
	CSV_DATA_EXCHANGER_SELECT_PATH					:= 60,
	CSV_DATA_EXCHANGER_CREATE_TABLE					:= 70,	
	CSV_DATA_EXCHANGER_INSERT_INTO_TABLE			:= 80,	(* Writting logs to file *)
	CSV_DATA_EXCHANGER_RESET 						:= 90,	(* Reseting function block *)
	CSV_DATA_EXCHANGER_METHOD_DONE					:= 100,	(* Writting done *)
	CSV_DATA_EXCHANGER_ABORTING						:= -10	(* Aborting *)
);
END_TYPE

// ---- DUTs/Libs/Utilities/CSV Data Exchanger/ST_CSV_Record.TcDUT
TYPE ST_CSV_Record :
STRUCT
	sName 	: T_MaxString 	:= '';
	nNumber	: UDINT 		:= 0;
	fPos	: LREAL 		:= 0.0;
	bOP		: BOOL 			:= FALSE;
	sDesc	: STRING(40)	:= '';
	data	: ARRAY[0..7] OF BYTE;
END_STRUCT
END_TYPE

// ---- DUTs/Libs/Utilities/File Logger/E_FileLoggerAddLogsState.TcDUT
{attribute 'strict'}
TYPE E_FileLoggerAddLogsState :
(
	FILE_LOGGER_ADD_LOGS_OPEN 			:= 0,	(* Opening file *)
	FILE_LOGGER_ADD_LOGS_WRITTE			:= 10,	(* Writting log from buffer to file *)
	FILE_LOGGER_ADD_LOGS_WRITTE_DONE	:= 20,	(* Writting log from buffer to file done *)
	FILE_LOGGER_ADD_LOGS_CLOSE 			:= 30,	(* Closing file *)
	FILE_LOGGER_ADD_LOGS_CLEAR			:= 40	(* Clearing buffer *)
);
END_TYPE

// ---- DUTs/Libs/Utilities/File Logger/E_FileLoggerInitState.TcDUT
{attribute 'strict'}
TYPE E_FileLoggerInitState :
(
	FILE_LOGGER_INIT_CREATE_DIR 	:= 0,	(* Creating directory if doesn't exist *)
	FILE_LOGGER_INIT_GET_TIME		:= 10,	(* Getting current time *)
	FILE_LOGGER_INIT_CREATE_FILE	:= 20,	(* Creating empty file of logger *)
	FILE_LOGGER_INIT_ADD_HEADER		:= 30,	(* Adding header at the beggining of file *)
	FILE_LOGGER_INIT_CLOSE_FILE		:= 40,	(* Closing file *)
	FILE_LOGGER_INIT_DONE 			:= 50	(* Initiazlization done *)
);
END_TYPE

// ---- DUTs/Libs/Utilities/File Logger/E_FileLoggerSetNewPathState.TcDUT
{attribute 'strict'}
TYPE E_FileLoggerSetNewPathState :
(
	FILE_LOGGER_SET_NEW_PATH_CHANGE_PATH			:= 0,
	FILE_LOGGER_SET_NEW_PATH_DONE					:= 10
);
END_TYPE

// ---- DUTs/Libs/Utilities/File Logger/E_FileLoggerState.TcDUT
{attribute 'strict'}
TYPE E_FileLoggerState :
(
	FILE_LOGGER_UNINITIALIZED 	:= 0,	(* Not ready to work *)
	FILE_LOGGER_INITIALIZING	:= 10,	(* Preparing to work *)
	FILE_LOGGER_READY 			:= 20,	(* Ready ti work, waiting for logs in buffer *)
	FILE_LOGGER_IDLE 			:= 30,	(* Ready ti work, waiting for logs in buffer *)
	FILE_LOGGER_ADD_LOGS		:= 40,	(* Writting logs to file *)
	FILE_LOGGER_SELECT_PATH		:= 50,	(* Writting done *)
	FILE_LOGGER_RESET 			:= 60,	(* Reseting function block *)
	FILE_LOGGER_METHOD_DONE		:= 70,	(* Reseting done *)
	FILE_LOGGER_ABORTING		:= -10	(* Aborting *)
);
END_TYPE

// ---- DUTs/Libs/Utilities/Recipe Manager/E_RecipesManagerReturns.TcDUT
{attribute 'strict'}
TYPE E_RecipesManagerReturns :
(
	RECIPES_MANAGER_ERR_OK										:= 0,	(* The operation was carried out successfully *)
	RECIPES_MANAGER_ERR_FAILED									:= 10,	(* The operation failed *)
	RECIPES_MANAGER_ERR_PARAMETER								:= 20,	(* Incorrect parameter *)
	RECIPES_MANAGER_ERR_NOTINITALIZED							:= 30,	(* The data server object is not initialized *)
	RECIPES_MANAGER_ERR_NOIMPLEMENTED							:= 40,	(* The data server does not implement *)
	RECIPES_MANAGER_ERR_NO_OBJECT								:= 50,	(* Not all variables of a recipe definition can be written via the data server *)
	RECIPES_MANAGER_ERR_NOMEMORY								:= 60,	(* The recipe definition has no free memory to create a new recipe *)
	RECIPES_MANAGER_ERR_RECIPE_FILE_NOT_FOUND 					:= 70,	(* The recipe file was not found *)
	RECIPES_MANAGER_ERR_RECIPE_MISMATCH							:= 80,	(* The contents of the recipe file do not match the current recipe *)
	RECIPES_MANAGER_ERR_RECIPE_SAVE_ERR							:= 90,	(* The storage procedure failed *)
	RECIPES_MANAGER_ERR_RECIPE_NOT_FOUND						:= 100,	(* The recipe does not exist *)
	RECIPES_MANAGER_ERR_RECIPE_DEFINITION_NOT_FOUND				:= 110,	(* The recipe definition does not exist *)
	RECIPES_MANAGER_ERR_RECIPE_ALREADY_EXIST					:= 120,	(* The recipe already exists in the recipe definition *)
	RECIPES_MANAGER_ERR_NO_RECIPE_MANAGER_SET					:= 130,	(* The global recipe manager has not been created *)
	RECIPES_MANAGER_ERR_RECIPE_NOT_ALL_VARIABLES_WERE_LOADED	:= 140,	(* The recipe definition contains more variables than the recipe file *)
	RECIPES_MANAGER_ERR_RECIPES_MANAGER_LOCKED					:= 150,	(* The recipe manager was blocked during the online change *)
	RECIPES_MANAGER_ERR_SOURCE_EXHAUSTED						:= 160,	(* Used for UTF8 Helper *)
	RECIPES_MANAGER_ERR_TARGET_EXHAUSTED						:= 170,	(* Used for UTF8 Helper *)
	RECIPES_MANAGER_ERR_SOURCE_ILLEGAL							:= 180	(* Used for UTF8 Helper *)
);
END_TYPE

// ---- DUTs/Libs/Utilities/Recipe Manager/E_RecipesManagerState.TcDUT
{attribute 'strict'}
TYPE E_RecipesManagerState :
(
	RECIPES_MANAGER_UNINITIALIZED					:= 0,	(* Not ready to work *)
	RECIPES_MANAGER_INITIALIZATION					:= 10,	(* Preparing to work *)
	RECIPES_MANAGER_IDLE							:= 20,	(* Waiting for commands *)
	RECIPES_MANAGER_CREATE							:= 30,	(* Creating new recipe definition *)
	RECIPES_MANAGER_CREATE_DONE						:= 40,	(* Creating new recipe definition done *)
	RECIPES_MANAGER_REMOVE							:= 50,	(* Removing recipe definition *)
	RECIPES_MANAGER_REMOVE_DONE						:= 60,	(* Removing recipe definition done *)
	RECIPES_MANAGER_LOAD							:= 70,	(* Loading recie from file to recipe manager *)
	RECIPES_MANAGER_LOAD_DONE						:= 80,	(* Loading done *)
	RECIPES_MANAGER_SAVE							:= 90,	(* Saving current recipe definition value from recipe manager to file *)
	RECIPES_MANAGER_SAVE_DONE						:= 100,	(* Saving done *)
	RECIPES_MANAGER_READ							:= 110,	(* Reading values from variable to recipe definition i recipe manager *)
	RECIPES_MANAGER_READ_DONE						:= 120,	(* Reding done *)
	RECIPES_MANAGER_READ_AND_SAVE					:= 130,	(* Reading and saving values from variable to file *)
	RECIPES_MANAGER_READ_AND_SAVE_DONE				:= 140,	(* Readin and saving done *)
	RECIPES_MANAGER_WRITE							:= 150,	(* Writing values from recipe definition in recipe manager to variables *)
	RECIPES_MANAGER_WRITE_DONE						:= 160,	(* Writing done *)
	RECIPES_MANAGER_LOAD_AND_WRITE					:= 170,	(* Loading values from file and writing to variables*)
	RECIPES_MANAGER_LOAD_AND_WRITE_DONE 			:= 180,	(* Loadind and writing done *)
	RECIPES_MANAGER_GET_RECIPE_NAME_ARRAY			:= 190,	(* Getting names of recipes in selected directory*)
	RECIPES_MANAGER_GET_RECIPE_NAME_ARRAY_DONE		:= 200,	(* Getting names of recipes done *)
	RECIPES_MANAGER_GET_RECIPE_VARIABLE_NAMES		:= 210, (* Getting names of variables from recipes manager *)
	RECIPES_MANAGER_GET_RECIPE_VARIABLE_NAMES_DONE	:= 220,	(* Getting names of variables done *)
	RECIPES_MANAGER_GET_RECIPE_VARIABLE_VALUES		:= 230,	(* Getting variable values from recipes files *)
	RECIPES_MANAGER_GET_RECIPE_VARIABLE_VALUES_DONE	:= 240,	(* Getting variables values done *)
	RECIPES_MANAGER_RELOAD							:= 250, (* Reload recipes manager *)
	RECIPES_MANAGER_RELOAD_DONE						:= 260,	(* Reload done *)
	RECIPES_MANAGER_BACKUP							:= 270,	(* Perform backup of all recipes to selected directory *)
	RECIPES_MANAGER_BACKUP_DONE						:= 280,	(* Backup done*)
	RECIPES_MANAGER_RESTORE							:= 290,	(* Restore recipes from selected directory *)
	RECIPES_MANAGER_RESTORE_DONE					:= 300,	(* Restoring done*)
	RECIPES_MANAGER_ABORTING						:= -10	(* Aborting *)
);
END_TYPE

// ---- DUTs/Libs/Utilities/Recipe Manager/E_RecipesManagerStateBackup.TcDUT
{attribute 'strict'}
TYPE E_RecipesManagerStateBackup :
(
	RECIPES_MANAGER_BACKUP_OPERATION 			:= 0,	(* Create/Remove recipe with selected name *)
	RECIPES_MANAGER_BACKUP_GET_RECIPES_COUNT 	:= 10,	(* Getting number of detected recipes in directory *)
	RECIPES_MANAGER_BACKUP_RELOAD				:= 20,	(* Reloading recipes manager *)
	RECIPES_MANAGER_BACKUP_GET_RECIPES_NAMES 	:= 30,	(* Getting names of recipes in selected directory *)
	RECIPES_MANAGER_BACKUP_GET_VARIABLE_NAMES	:= 40,	(* Getting names of variables from recipes manager *)
	RECIPES_MANAGER_BACKUP_GET_VARIABLE_VALUES	:= 50,	(* Getting variable values from selected recipe *)
	RECIPES_MANAGER_BACKUP_BACKUP_DONE			:= 60	(* Removing selected recipe *)

);
END_TYPE

// ---- DUTs/Libs/Utilities/Recipe Manager/E_RecipesManagerStateCreateRemove.TcDUT
{attribute 'strict'}
TYPE E_RecipesManagerStateCreateRemove :
(
	RECIPES_MANAGER_CREATE_REMOVE_OPERATION 			:= 0,	(* Create/Remove recipe with selected name *)
	RECIPES_MANAGER_CREATE_REMOVE_GET_RECIPES_COUNT 	:= 10,	(* Getting number of detected recipes in directory *)
	RECIPES_MANAGER_CREATE_REMOVE_RELOAD				:= 20,	(* Reloading recipes manager *)
	RECIPES_MANAGER_CREATE_REMOVE_GET_RECIPES_NAMES 	:= 30,	(* Getting names of recipes in selected directory *)
	RECIPES_MANAGER_CREATE_REMOVE_GET_VARIABLE_NAMES	:= 40,	(* Getting names of variables from recipes manager *)
	RECIPES_MANAGER_CREATE_REMOVE_GET_VARIABLE_VALUES	:= 50,	(* Getting variable values from selected recipe *)
	RECIPES_MANAGER_CREATE_REMOVE_DONE					:= 60	(* Removing selected recipe *)
);
END_TYPE

// ---- DUTs/Libs/Utilities/Recipe Manager/E_RecipesManagerStateInit.TcDUT
{attribute 'strict'}
TYPE E_RecipesManagerStateInit :
(
	RECIPES_MANAGER_INIT_SET_STORAGE_PATH 		:= 0,	(* Setting storage path *)
	RECIPES_MANAGER_INIT_RELOAD					:= 10,	(* Reloading recipes manager *)
	RECIPES_MANAGER_INIT_GET_RECIPES_COUNT		:= 20,	(* Getting number of detected recipes in directory *)
	RECIPES_MANAGER_INIT_GET_RECIPES_NAMES		:= 30,	(* Getting names of recipes in selected directory *)
	RECIPES_MANAGER_INIT_GET_VARIABLE_NAMES		:= 40,	(* Getting names of variables from recipes manager *)
	RECIPES_MANAGER_INIT_GET_VARIABLE_VALUES	:= 50,	(* Getting variable values from selected recipe *)
	RECIPES_MANAGER_INIT_DONE					:= 60,	(* Init procedure done *)
	RECIPES_MANAGER_INIT_ERROR					:= 255	(* Init procedure error*)
);
END_TYPE

// ---- DUTs/Libs/Utilities/Recipe Manager/E_RecipesManagerStateReload.TcDUT
{attribute 'strict'}
TYPE E_RecipesManagerStateReload :
(
	RECIPE_MANAGER_RELOAD_OPERATION 			:= 0,
	RECIPE_MANAGER_RELOAD_GET_RECIPES_COUNT 	:= 10,
	RECIPE_MANAGER_RELOAD_GET_RECIPES_NAMES 	:= 20,
	RECIPE_MANAGER_RELOAD_GET_VARIABLE_NAMES	:= 30,
	RECIPE_MANAGER_RELOAD_GET_VARIABLE_VALUES	:= 40,
	RECIPE_MANAGER_RELOAD_DONE					:= 50
);
END_TYPE

// ---- DUTs/Libs/Utilities/TXT Data Exchanger/E_TXTDataExchangerAddLogsState.TcDUT
{attribute 'strict'}
TYPE E_TXTDataExchangerAddLogsState :
(
	TXT_DATA_EXCHANGER_ADD_LOGS_OPEN 			:= 0,	(* Opening file *)
	TXT_DATA_EXCHANGER_ADD_LOGS_WRITE			:= 10,	(* Writting log from buffer to file *)
	TXT_DATA_EXCHANGER_ADD_LOGS_WRITE_DONE		:= 20,	(* Writting log from buffer to file done *)
	TXT_DATA_EXCHANGER_ADD_LOGS_CLOSE 			:= 30,	(* Closing file *)
	TXT_DATA_EXCHANGER_ADD_LOGS_CLEAR			:= 40	(* Clearing buffer *)
);
END_TYPE

// ---- DUTs/Libs/Utilities/TXT Data Exchanger/E_TXTDataExchangerInitState.TcDUT
{attribute 'strict'}
TYPE E_TXTDataExchangerInitState :
(
	TXT_DATA_EXCHANGER_INIT_CREATE_DIR 		:= 0,	(* Creating directory if doesn't exist *)
	TXT_DATA_EXCHANGER_INIT_GET_TIME		:= 10,	(* Getting current time *)
	TXT_DATA_EXCHANGER_INIT_CREATE_FILE		:= 20,	(* Creating empty file of logger *)
	TXT_DATA_EXCHANGER_INIT_ADD_HEADER		:= 30,	(* Adding header at the beggining of file *)
	TXT_DATA_EXCHANGER_INIT_CLOSE_FILE		:= 40,	(* Closing file *)
	TXT_DATA_EXCHANGER_INIT_DONE 			:= 50	(* Initiazlization done *)
);
END_TYPE

// ---- DUTs/Libs/Utilities/TXT Data Exchanger/E_TXTDataExchangerSearchForFileState.TcDUT
{attribute 'strict'}
TYPE E_TXTDataExchangerSearchForFileState :
(
	TXT_DATA_EXCHANGER_SEARCH_FOR_FILE_ENUM_FIRST_ENTRY			:= 0,
	TXT_DATA_EXCHANGER_SEARCH_FOR_FILE_ENUM_NEXT_ENTRY			:= 10,
	TXT_DATA_EXCHANGER_SEARCH_FOR_FILE_WAIT_FOR_READING			:= 20,
	TXT_DATA_EXCHANGER_SEARCH_FOR_FILE_DONE						:= 30
);
END_TYPE

// ---- DUTs/Libs/Utilities/TXT Data Exchanger/E_TXTDataExchangerSetNewPathState.TcDUT
{attribute 'strict'}
TYPE E_TXTDataExchangerSetNewPathState :
(
	TXT_DATA_EXCHANGER_SET_NEW_PATH_CHANGE_PATH			:= 0,
	TXT_DATA_EXCHANGER_SET_NEW_PATH_DONE				:= 10
);
END_TYPE

// ---- DUTs/Libs/Utilities/TXT Data Exchanger/E_TXTDataExchangerState.TcDUT
{attribute 'strict'}
TYPE E_TXTDataExchangerState :
(
	TXT_DATA_EXCHANGER_UNINITIALIZED 	:= 0,	(* Not ready to work *)
	TXT_DATA_EXCHANGER_INITIALIZING		:= 10,	(* Preparing to work *)
	TXT_DATA_EXCHANGER_READY 			:= 20,	(* Ready ti work, waiting for logs in buffer *)
	TXT_DATA_EXCHANGER_IDLE 			:= 30,	(* Ready ti work, waiting for logs in buffer *)
	TXT_DATA_EXCHANGER_ADD_LOGS			:= 40,	(* Writting logs to file *)
	TXT_DATA_EXCHANGER_SELECT_PATH		:= 50,	(* Writting done *)
	TXT_DATA_EXCHANGER_SEARCH_FOR_FILE	:= 60,	(* Writting done *)
	TXT_DATA_EXCHANGER_RESET 			:= 70,	(* Reseting function block *)
	TXT_DATA_EXCHANGER_METHOD_DONE		:= 80,	(* Reseting done *)
	TXT_DATA_EXCHANGER_ABORTING			:= -10	(* Aborting *)
);
END_TYPE

// ---- DUTs/Libs/Vision/Cognex/E_CognexCameraGetConnectionStatus.TcDUT
{attribute 'strict'}
TYPE E_CognexCameraGetConnectionStatus :
(
	WAITING_FOR_STATUS_CODE						:= 2,
	THE_COMMAND_WAS_EXECUTED_SUCCESSFULLY		:= 1,
	UNRECOGNIZED_COMMAND 						:= 0,
	THE_CELL_ID_IS_INVALID						:= -1,
	THE_COMMAND_COULD_NOT_BE_EXECUTED 			:= -2,
	USER_DOES_NOT_HAVE_FULL_ACCESS				:= -6
);
END_TYPE

// ---- DUTs/Libs/Vision/Cognex/E_CognexCameraGetExprStatus.TcDUT
{attribute 'strict'}
TYPE E_CognexCameraGetExprStatus :
(
	WAITING_FOR_STATUS_CODE										:= 2,
	THE_COMMAND_WAS_EXECUTED_SUCCESSFULLY						:= 1,
	UNRECOGNIZED_COMMAND 										:= 0,
	THE_CELL_ID_IS_INVALID_OR_HAS_EXCEEDED_15_BYTES_IN_LENGTH	:= -1,
	THE_COMMAND_COULD_NOT_BE_EXECUTED 							:= -2
);
END_TYPE

// ---- DUTs/Libs/Vision/Cognex/E_CognexCameraGetFileListStatus.TcDUT
{attribute 'strict'}
TYPE E_CognexCameraGetFileListStatus :
(
	WAITING_FOR_STATUS_CODE									:= 2,
	THE_COMMAND_WAS_EXECUTED_SUCCESSFULLY					:= 1,
	UNRECOGNIZED_COMMAND 									:= 0,
	THE_INPUT_IS_INVALID_OR_HAS_EXCEEDED_15_BYTES_IN_LENGTH	:= -1,
	THE_ACTIVE_JOB_HAS_NOT_BEEN_SAVED 						:= -2
);
END_TYPE

// ---- DUTs/Libs/Vision/Cognex/E_CognexCameraGetFileStatus.TcDUT
{attribute 'strict'}
TYPE E_CognexCameraGetFileStatus :
(
	WAITING_FOR_STATUS_CODE						:= 2,
	THE_COMMAND_WAS_EXECUTED_SUCCESSFULLY		:= 1,
	UNRECOGNIZED_COMMAND 						:= 0,
	THE_ACTIVE_JOB_HAS_NOT_BEEN_SAVED 			:= -2
);
END_TYPE

// ---- DUTs/Libs/Vision/Cognex/E_CognexCameraGetJobStatus.TcDUT
{attribute 'strict'}
TYPE E_CognexCameraGetJobStatus :
(
	WAITING_FOR_STATUS_CODE														:= 2,
	THE_COMMAND_WAS_EXECUTED_SUCCESSFULLY										:= 1,
	UNRECOGNIZED_COMMAND 														:= 0,
	THE_ACTIVE_JOB_HAS_NOT_BEEN_SAVED_OR_DOES_NOT_HAVE_A_NUMERICAL_PREFIX		:= -2
);
END_TYPE

// ---- DUTs/Libs/Vision/Cognex/E_CognexCameraGetOnlineStatus.TcDUT
{attribute 'strict'}
TYPE E_CognexCameraGetOnlineStatus :
(
	WAITING_FOR_STATUS_CODE								:= 2,
	THE_IN_SIGHT_VISION_SYSTEM_IS_CURRENTLY_OFFLINE		:= 0,
	THE_IN_SIGHT_VISION_SYSTEM_IS_CURRENTLY_ONLINE 		:= 1
);
END_TYPE

// ---- DUTs/Libs/Vision/Cognex/E_CognexCameraGetPositionState.TcDUT
{attribute 'strict'}
TYPE E_CognexCameraGetPositionState :
(
	CAMERA_GET_POSITION_SEND_COMMAND_X				:= 0,
	CAMERA_GET_POSITION_RECEIVE_RESPONSE_X			:= 10,
	CAMERA_GET_POSITION_SEND_COMMAND_Y				:= 20,
	CAMERA_GET_POSITION_RECEIVE_RESPONSE_Y			:= 30,
	CAMERA_GET_POSITION_SEND_COMMAND_ROTATION		:= 40,
	CAMERA_GET_POSITION_RECEIVE_RESPONSE_ROTATION	:= 50,
	CAMERA_GET_POSITION_GETTING_DONE				:= 60
);
END_TYPE

// ---- DUTs/Libs/Vision/Cognex/E_CognexCameraGetPositionStatus.TcDUT
{attribute 'strict'}
TYPE E_CognexCameraGetPositionStatus :
(
	WAITING_FOR_STATUS_CODE						:= 2,
	THE_COMMAND_WAS_EXECUTED_SUCCESSFULLY		:= 1,
	UNRECOGNIZED_COMMAND 						:= 0,
	THE_SYMBOLIC_TAG_IS_INVALID					:= -1,
	THE_COMMAND_COULD_NOT_BE_EXECUTED 			:= -2,
	PRODUCT_NOT_FOUND							:= -3
);
END_TYPE

// ---- DUTs/Libs/Vision/Cognex/E_CognexCameraGetValueEasyBuilderStatus.TcDUT
{attribute 'strict'}
TYPE E_CognexCameraGetValueEasyBuilderStatus :
(
	WAITING_FOR_STATUS_CODE						:= 2,
	THE_COMMAND_WAS_EXECUTED_SUCCESSFULLY		:= 1,
	UNRECOGNIZED_COMMAND 						:= 0,
	THE_SYMBOLIC_TAG_IS_INVALID					:= -1,
	THE_COMMAND_COULD_NOT_BE_EXECUTED 			:= -2
);
END_TYPE

// ---- DUTs/Libs/Vision/Cognex/E_CognexCameraGetValueSpreadsheetStatus.TcDUT
{attribute 'strict'}
TYPE E_CognexCameraGetValueSpreadsheetStatus :
(
	WAITING_FOR_STATUS_CODE						:= 2,
	THE_COMMAND_WAS_EXECUTED_SUCCESSFULLY		:= 1,
	UNRECOGNIZED_COMMAND 						:= 0,
	THE_CELL_ID_IS_INVALID						:= -1,
	THE_COMMAND_COULD_NOT_BE_EXECUTED 			:= -2
);
END_TYPE

// ---- DUTs/Libs/Vision/Cognex/E_CognexCameraGetValuesState.TcDUT
{attribute 'strict'}
TYPE E_CognexCameraGetValuesState :
(
	CAMERA_GET_VALUES_SEND_COMMAND_VALUE_1		:= 0,
	CAMERA_GET_VALUES_RECEIVE_RESPONSE_VALUE_1	:= 10,
	CAMERA_GET_VALUES_SEND_COMMAND_VALUE_2		:= 20,
	CAMERA_GET_VALUES_RECEIVE_RESPONSE_VALUE_2	:= 30,
	CAMERA_GET_VALUES_SEND_COMMAND_VALUE_3		:= 40,
	CAMERA_GET_VALUES_RECEIVE_RESPONSE_VALUE_3	:= 50,
	CAMERA_GET_VALUES_SEND_COMMAND_VALUE_4		:= 60,
	CAMERA_GET_VALUES_RECEIVE_RESPONSE_VALUE_4	:= 70,
	CAMERA_GET_VALUES_GETTING_DONE				:= 80
);
END_TYPE

// ---- DUTs/Libs/Vision/Cognex/E_CognexCameraGetValuesStatus.TcDUT
{attribute 'strict'}
TYPE E_CognexCameraGetValuesStatus :
(
	WAITING_FOR_STATUS_CODE						:= 2,
	THE_COMMAND_WAS_EXECUTED_SUCCESSFULLY		:= 1,
	UNRECOGNIZED_COMMAND 						:= 0,
	THE_SYMBOLIC_TAG_IS_INVALID					:= -1,
	THE_COMMAND_COULD_NOT_BE_EXECUTED 			:= -2,
	ONE_OR_MORE_VALUE_IS_INVALID				:= -3
);
END_TYPE

// ---- DUTs/Libs/Vision/Cognex/E_CognexCameraGetValueStatus.TcDUT
{attribute 'strict'}
TYPE E_CognexCameraGetValueStatus :
(
	WAITING_FOR_STATUS_CODE						:= 2,
	THE_COMMAND_WAS_EXECUTED_SUCCESSFULLY		:= 1,
	UNRECOGNIZED_COMMAND 						:= 0,
	THE_CELL_ID_IS_INVALID						:= -1,
	THE_COMMAND_COULD_NOT_BE_EXECUTED 			:= -2,
	USER_DOES_NOT_HAVE_FULL_ACCESS				:= -6
);
END_TYPE

// ---- DUTs/Libs/Vision/Cognex/E_CognexCameraImageTriggerStatus.TcDUT
{attribute 'strict'}
TYPE E_CognexCameraImageTriggerStatus :
(
	WAITING_FOR_STATUS_CODE										:= 2,
	THE_COMMAND_WAS_EXECUTED_SUCCESSFULLY						:= 1,
	UNRECOGNIZED_COMMAND 										:= 0,
	THE_NUMBER_IS_EITHER_OUT_OF_RANGE_OR_NOT_AN_INTEGER 		:= -1,
	THE_COMMAND_COULD_NOT_BE_EXECUTED_OR_THE_SENSOR_IS_OFFLINE 	:= -2,
	USER_DOES_NOT_HAVE_FULL_ACCESS								:= -6
);
END_TYPE

// ---- DUTs/Libs/Vision/Cognex/E_CognexCameraInitState.TcDUT
{attribute 'strict'}
TYPE E_CognexCameraInitState :
(
	CAMERA_INIT_CONNECTION 				:= 0,
	CAMERA_INIT_CLEAR_BUFFER			:= 10,	
	CAMERA_INIT_WAIT_FOR_USERNAME 		:= 20,	
	CAMERA_INIT_WRITE_USER				:= 30,	
	CAMERA_INIT_WAIT_FOR_PASSWORD 		:= 40,	
	CAMERA_INIT_WRITE_PASSWORD			:= 50,	
	CAMERA_INIT_WAIT_FOR_CONFIRMATION	:= 60,
	CAMERA_INIT_DONE					:= 80
);
END_TYPE

// ---- DUTs/Libs/Vision/Cognex/E_CognexCameraLoadFileStatus.TcDUT
{attribute 'strict'}
TYPE E_CognexCameraLoadFileStatus :
(
	WAITING_FOR_STATUS_CODE						:= 2,
	THE_COMMAND_WAS_EXECUTED_SUCCESSFULLY		:= 1,
	UNRECOGNIZED_COMMAND 						:= 0,
	THE_FILENAME_IS_MISSING						:= -1,
	THE_JOB_FAILED_TO_LOAD 						:= -2,
	THE_VISION_SYSTEM_IS_OUT_OF_MEMORY			:= -4,
	USER_DOES_NOT_HAVE_FULL_ACCESS				:= -6
);
END_TYPE

// ---- DUTs/Libs/Vision/Cognex/E_CognexCameraMethodState.TcDUT
{attribute 'strict'}
TYPE E_CognexCameraMethodState :
(
	CAMERA_METHOD_SEND_COMMAND 			:= 0,
	CAMERA_METHOD_RECEIVE_RESPONSE 		:= 10
);
END_TYPE

// ---- DUTs/Libs/Vision/Cognex/E_CognexCameraPutLiveStatus.TcDUT
{attribute 'strict'}
TYPE E_CognexCameraPutLiveStatus :
(
	WAITING_FOR_STATUS_CODE										:= 2,
	THE_COMMAND_WAS_EXECUTED_SUCCESSFULLY						:= 1,
	UNRECOGNIZED_COMMAND 										:= 0,
	THE_INPUT_IS_INVALID_OR_HAS_EXCEEDED_15_BYTES_IN_LENGTH		:= -1,
	THE_COMMAND_COULD_NOT_BE_EXECUTED 							:= -2,
	USER_DOES_NOT_HAVE_FULL_ACCESS	 							:= -6
);
END_TYPE

// ---- DUTs/Libs/Vision/Cognex/E_CognexCameraPutPortnumStatus.TcDUT
{attribute 'strict'}
TYPE E_CognexCameraPutPortnumStatus :
(
	WAITING_FOR_STATUS_CODE										:= 2,
	THE_COMMAND_WAS_EXECUTED_SUCCESSFULLY						:= 1,
	UNRECOGNIZED_COMMAND 										:= 0,
	THE_INPUT_IS_INVALID_OR_HAS_EXCEEDED_15_BYTES_IN_LENGTH		:= -1,
	THE_COMMAND_COULD_NOT_BE_EXECUTED 							:= -2,
	USER_DOES_NOT_HAVE_FULL_ACCESS	 							:= -6
);
END_TYPE

// ---- DUTs/Libs/Vision/Cognex/E_CognexCameraPutTimeoutStatus.TcDUT
{attribute 'strict'}
TYPE E_CognexCameraPutTimeoutStatus :
(
	WAITING_FOR_STATUS_CODE										:= 2,	
	THE_COMMAND_WAS_EXECUTED_SUCCESSFULLY						:= 1,
	UNRECOGNIZED_COMMAND 										:= 0,
	THE_INPUT_IS_INVALID_OR_HAS_EXCEEDED_15_BYTES_IN_LENGTH		:= -1,
	USER_DOES_NOT_HAVE_FULL_ACCESS	 							:= -6
);
END_TYPE

// ---- DUTs/Libs/Vision/Cognex/E_CognexCameraPutUpdateStatus.TcDUT
{attribute 'strict'}
TYPE E_CognexCameraPutUpdateStatus :
(
	WAITING_FOR_STATUS_CODE										:= 2,	
	THE_COMMAND_WAS_EXECUTED_SUCCESSFULLY						:= 1,
	UNRECOGNIZED_COMMAND 										:= 0,
	THE_INPUT_IS_INVALID_OR_HAS_EXCEEDED_15_BYTES_IN_LENGTH		:= -1,
	THE_COMMAND_COULD_NOT_BE_EXECUTED 							:= -2,
	USER_DOES_NOT_HAVE_FULL_ACCESS	 							:= -6
);
END_TYPE

// ---- DUTs/Libs/Vision/Cognex/E_CognexCameraPutWatchStatus.TcDUT
{attribute 'strict'}
TYPE E_CognexCameraPutWatchStatus :
(
	WAITING_FOR_STATUS_CODE										:= 2,	
	THE_COMMAND_WAS_EXECUTED_SUCCESSFULLY						:= 1,
	UNRECOGNIZED_COMMAND 										:= 0,
	THE_INPUT_IS_INVALID_OR_HAS_EXCEEDED_15_BYTES_IN_LENGTH		:= -1,
	THE_COMMAND_COULD_NOT_BE_EXECUTED 							:= -2,
	USER_DOES_NOT_HAVE_FULL_ACCESS								:= -6
);
END_TYPE

// ---- DUTs/Libs/Vision/Cognex/E_CognexCameraResetSystemStatus.TcDUT
{attribute 'strict'}
TYPE E_CognexCameraResetSystemStatus :
(
	WAITING_FOR_STATUS_CODE					:= 2,	
	THE_COMMAND_WAS_EXECUTED_SUCCESSFULLY	:= -1,
	USER_DOES_NOT_HAVE_FULL_ACCESS			:= -6
);
END_TYPE

// ---- DUTs/Libs/Vision/Cognex/E_CognexCameraSetJobStatus.TcDUT
{attribute 'strict'}
TYPE E_CognexCameraSetJobStatus :
(
	WAITING_FOR_STATUS_CODE														:= 2,	
	THE_COMMAND_WAS_EXECUTED_SUCCESSFULLY										:= 1,
	UNRECOGNIZED_COMMAND 														:= 0,
	THE_ID_IS_LESS_THAN_0_OR_IS_NOT_AN_INTEGER									:= -1,
	THE_JOB_FAILED_TO_LOAD_THE_SENSOR_IS_ONLINE_OR_THE_FILE_WAS_NOT_FOUND		:= -2,
	THE_IN_SIGHT_SENSOR_IS_OUT_OF_MEMORY										:= -4,
	USER_DOES_NOT_HAVE_FULL_ACCESS												:= -6
);
END_TYPE

// ---- DUTs/Libs/Vision/Cognex/E_CognexCameraSetOnlineStatus.TcDUT
{attribute 'strict'}
TYPE E_CognexCameraSetOnlineStatus :
(
	WAITING_FOR_STATUS_CODE																		:= 2,	
	THE_COMMAND_WAS_EXECUTED_SUCCESSFULLY														:= 1,
	UNRECOGNIZED_COMMAND 																		:= 0,
	THE_VALUE_GIVEN_FOR_INT_IS_EITHER_OUT_OF_RANGE_OR_IS_NOT_A_VALID_INTEGER					:= -1,
	THE_COMMAND_COULD_NOT_BE_EXECUTED 															:= -2,
	THE_SENSOR_DID_NOT_GO_ONLINE_BECAUSE_IS_SET_OFFLINE_MANUAL_OR_BY_A_DISCRETE_IO_SIGNAL		:= -5,
	USER_DOES_NOT_HAVE_FULL_ACCESS																:= -6
);
END_TYPE

// ---- DUTs/Libs/Vision/Cognex/E_CognexCameraState.TcDUT
{attribute 'strict'}
TYPE E_CognexCameraState :
(
	CAMERA_UNINITIALIZED 				:= 0,	(* Not ready to work *)
	CAMERA_INITIALIZING					:= 10,	(* Preparing to work *)
	CAMERA_READY 						:= 20,	(* Ready to work *)
	CAMERA_IDLE							:= 30,	(* Waiting for commands *)
	CAMERA_RESET 						:= 40,	(* Reseting function block *)
	CAMERA_LOAD_FILE					:= 50,
	CAMERA_GET_FILE						:= 60,
	CAMERA_GET_VALUE_EASY_BUILDER		:= 70,
	CAMERA_GET_VALUE_SPREADSHEET		:= 80,
	CAMERA_SET_ONLINE					:= 90,
	CAMERA_GET_ONLINE					:= 100,
	CAMERA_RESET_SYSTEM					:= 110,
	CAMERA_GET_CONNECTIONS				:= 120,
	CAMERA_GET_EXPR						:= 130,
	CAMERA_GET_FILE_LIST				:= 140,
	CAMERA_PUT_LIVE						:= 150,
	CAMERA_PUT_PORTNUM					:= 160,
	CAMERA_PUT_TIMEOUT					:= 170,
	CAMERA_PUT_UPDATE					:= 180,
	CAMERA_PUT_WATCH					:= 190,
	CAMERA_SET_JOB						:= 200,
	CAMERA_GET_JOB						:= 210,
	CAMERA_STORE_FILE					:= 220,
	CAMERA_GET_POSITION					:= 230,
	CAMERA_IMAGE_TRIGGER				:= 240,
	CAMERA_GET_VALUES					:= 250,
	CAMERA_METHOD_DONE					:= 260,
	CAMERA_ABORTING						:= -10	(* Aborting *)
);
END_TYPE

// ---- DUTs/Libs/Vision/Cognex/E_CognexCameraStoreFileStatus.TcDUT
{attribute 'strict'}
TYPE E_CognexCameraStoreFileStatus :
(
	WAITING_FOR_STATUS_CODE																	:= 2,	
	THE_COMMAND_WAS_EXECUTED_SUCCESSFULLY													:= 1,
	UNRECOGNIZED_COMMAND 																	:= 0,
	THE_FILENAME_IS_MISSING																	:= -1,
	THE_JOB_FAILED_TO_SAVE_THE_VISION_SYSTEM_IS_ONLINE_OR_THE_FILE_WAS_NOT_FOUND 			:= -2,
	USER_DOES_NOT_HAVE_FULL_ACCESS															:= -6
);
END_TYPE

// ---- DUTs/Machine/Machine Control/E_MachineCtrlStateInit.TcDUT
{attribute 'strict'}
TYPE E_MachineCtrlStateInit :
(	
	(* Robot init *)                                          		
	MACHINE_STATE_INITIALIZING_ROBOT_ABORT						:= 0,	(*  *)
	MACHINE_STATE_INITIALIZING_ROBOT_INIT						:= 10,	(*  *)
	MACHINE_STATE_INITIALIZING_ROBOT_HOME						:= 20,	(*  *)
	MACHINE_STATE_INITIALIZING_ROBOT_AUTOMATIC_MODE				:= 30,	(*  *)
                       	
	MACHINE_STATE_INITIALIZING_DONE								:= 40	(*  *)
)UINT;
END_TYPE

// ---- DUTs/Machine/Machine Control/E_MachineCtrlStateUninitialized.TcDUT
{attribute 'strict'}
TYPE E_MachineCtrlStateUninitialized :
(
	MACHINE_STATE_UNINITIALIZED_CR800_ETHERCAT_STATUS_CHECK 		:= 0,
	MACHINE_STATE_UNINITIALIZED_CR800_ETHERCAT_STATUS_CHECK_DONE	:= 10,
	MACHINE_STATE_UNINITIALIZED_CR800_ETHERCAT_ERROR_RESET			:= 20,
	MACHINE_STATE_UNINITIALIZED_CR800_ETHERCAT_REQUEST_OP_STATE		:= 30,	(*  *)
	MACHINE_STATE_UNINITIALIZED_CR800_CHECK_POWER_REGISTER			:= 40,	(*  *)
	MACHINE_STATE_UNINITIALIZED_DONE								:= 50	(*  *)
);
END_TYPE

// ---- DUTs/Machine/Shell API/ST_Shell.TcDUT
TYPE ST_Shell :
STRUCT
	stPlatform		: ST_ShellPlatform;		(*  *)
	stFlags			: ST_ShellFlags;		(*  *)
	stRecipeData	: ST_ShellRecipeData;	(*  *)
END_STRUCT
END_TYPE

// ---- DUTs/Machine/Shell API/ST_ShellFlags.TcDUT
TYPE ST_ShellFlags :
STRUCT
	bMachineCtrlAssignamentsDone	: BOOL := FALSE;	(*  *)
	bVisuCtrlAssignamentsDone		: BOOL := FALSE;	(*  *)
	bAlarmCtrlAssignamentsDone		: BOOL := FALSE;	(*  *)
	bRecipesCtrlAssignamentsDone	: BOOL := FALSE;	(*  *)
END_STRUCT
END_TYPE

// ---- DUTs/Machine/Shell API/ST_ShellPlatform.TcDUT
TYPE ST_ShellPlatform EXTENDS ST_UniversalPlatform :
STRUCT
	ref_fbMachineControler : REFERENCE TO FB_MachineControl;	(*  *)
	//refFbMachineSafety	: REFERENCE TO FB_MachineSafety;	(*  *)
	ref_fbVisuControler	: REFERENCE TO FB_VisuControl;			(*  *)
END_STRUCT
END_TYPE

// ---- DUTs/Machine/Shell API/ST_ShellRecipeData.TcDUT
TYPE ST_ShellRecipeData :
STRUCT
	(* Add recipe variables here and link them with RecipeManager in Tc3 XAE Shell *)
	rpVar1 : FB_RecipeParameter;
	rpVar2 : FB_RecipeParameter;
	rpVar3 : FB_RecipeParameter;
	rpVar4 : FB_RecipeParameter;
	rpVar5 : FB_RecipeParameter;
	rpVar6 : FB_RecipeParameter;
	rpVar7 : FB_RecipeParameter;
	rpVar8 : FB_RecipeParameter;
	rpVar9 : FB_RecipeParameter;
    rpVar10 : FB_RecipeParameter;
END_STRUCT
END_TYPE

// ---- GVLs/GVL.TcGVL
VAR_GLOBAL CONSTANT	
	(* --- Alarm controler --- *)
	iMAX_DEFINITION_EVENTS					: UDINT := 512; 													(* Maximum size of active alarms table *)
	iMAX_EVENTS								: UDINT	:= 512; 													(* Maximum size of events table *) 
	
	(* --- Recipes manager --- *)
	iMAX_NUMBER_OF_RECIPES					: USINT 		:= 128;												(* Defines maximum number of recipes stored in recipe manager *)
	iMAX_NUMBER_OF_VARIABLES_IN_RECIPES		: USINT			:= 128;												(* Defines maximum number of parameters stored inside the recipe *)
	iMAX_RECIPE_NAME_LENGTH					: INT			:= 80;												(* Defines maximum length of the recipe name *)
	iMAX_RECIPE_DESCRIPTION_LENGTH			: INT			:= 1024;											(* Defines maximum length of the recipe description on HMI screen *)
	iMAX_RECIPE_RESTOR_BACKUP_PATH_LENGTH	: INT			:= 1024;											(* Defines maximum lenght of the path where recipes are backuped/restored *)
	sDEFAULT_RECIPE_DEFINITON				: STRING		:= 'Recipes';										(* Defines default name of recipe definition inside recipe manager *)
	sDEFAULT_LOCAL_STORAGE_PATH				: STRING(512)	:= 'C:\TwinCAT\Tests\Recipes\';						(* Defines defaul path of recipe storage *)
	
